(* Logix 5000 project; controller PBS_Perfusion vendor 1 type 14 code 217 rev 32.14; software revision 32.03; part 5 of 27 *)
(* tags used below, declared in another part *)
   ONS : DINT[3];
   P101 : P_VSD;   // Feed Pump
   P103 : P_VSD;   // Conditioned Media Addition Pump
   P104 : P_VSD;   // Recirculation Pump
   P105 : P_VSD;   // Spent Media Pump
   REAL : DINT;

ADD_ON_INSTRUCTION AMP_Update_Jog_Speed   (* revision 1.0 *)
// Applied Motion - Update Jog Speed AOI
// Help:
// The Jog Move AOI is used to start jogging an axis at a specified speed and direction (a negative speed set point implies a CCW direction).
VAR_IN_OUT
   Input : DINT[14]; {required}   // Drive Input Assembly
   Output : DINT[16]; {required}   // Drive Output Assembly
        [0]   // Command Word
        [1]   // Jog Speed (0.25 rev/min)
        [2]   // Jog Acceleration (10 rev/s/s)
        [3]   // Jog Deceleration (10 rev/s/s)
        [4]   // Point-to-Point Velocity (0.25 rev/min)
        [5]   // Point-to-Point Acceleration (10 rev/min/s)
        [6]   // Point-to-Point Deceleration (10 rev/min/s)
        [7]   // Point-to-Point Distance (Motor steps)
        [9]   // (2x ASCII Letters in 16 lower word)
        [10]   // Data/Register 1
        [11]   // Data/Register 2
END_VAR
VAR_INPUT
   RPI : DINT := 100; {visible}   // Drive Connection Request Packet Interval (milliseconds)
   Start : BOOL; {required}   // Start the Relative Move
   Speed : REAL; {required}   // Updated Jog Velocity (rev/min)
END_VAR
VAR_OUTPUT
   Sent : BOOL; {access Read Only, visible}   // Updated Jog Velocity has been sent to drive
   In_Progress : BOOL; {access Read Only, visible}   // Jog Velocity Update in progress
   Done : BOOL; {access Read Only, visible}   // Jog Velocity Update completed without errors
   Error : BOOL; {access Read Only, visible}   // Jog Velocity Update failed to complete - drive not ready or faulted
   State : DINT := 10; {access Read Only}   // Internal state of progress
END_VAR
VAR
   Loc_StatusCode : AMP_Status_Word;
   Loc_CommandOff_Timer : TIMER;   // Timer to make sure command value was 0 before sending a new command
   Loc_CommandOn_Timer : TIMER;   // Timer to make sure command value is set long enough to be sent to drive
   Loc_Input_Assembly : AMP_Input_Assembly_v2; {access None}
   Loc_Start_ONS : BOOL; {access None}
   Loc_AlarmCode : AMP_Alarm_Word; {access None}
END_VAR

ROUTINE Logic   (* ladder *)
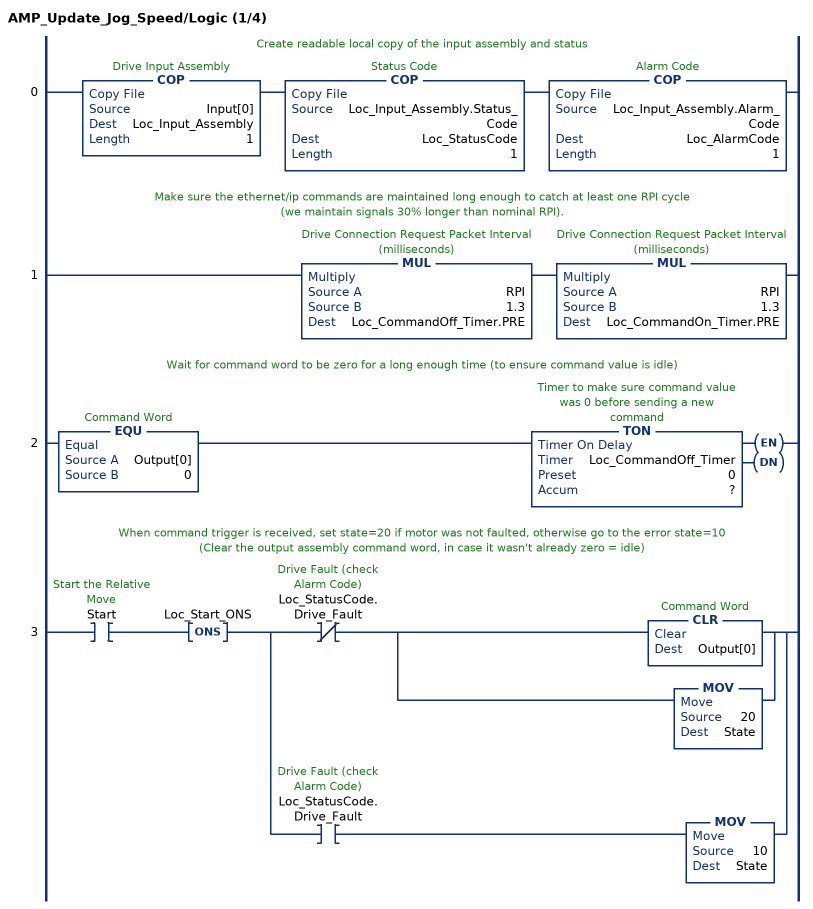
   // Create readable local copy of the input assembly and status
   0: COP(Input[0],Loc_Input_Assembly,1)COP(Loc_Input_Assembly.Status_Code,Loc_StatusCode,1)COP(Loc_Input_Assembly.Alarm_Code,Loc_AlarmCode,1);
   // Make sure the ethernet/ip commands are maintained long enough to catch at least one RPI cycle
   // (we maintain signals 30% longer than nominal RPI).
   1: MUL(RPI,1.3,Loc_CommandOff_Timer.PRE)MUL(RPI,1.3,Loc_CommandOn_Timer.PRE);
   // Wait for command word to be zero for a long enough time (to ensure command value is idle)
   2: EQU(Output[0],0)TON(Loc_CommandOff_Timer,?,?);
   // When command trigger is received, set state=20 if motor was not faulted, otherwise go to the error state=10
   // (Clear the output assembly command word, in case it wasn't already zero = idle)
   3: XIC(Start)ONS(Loc_Start_ONS)[XIO(Loc_StatusCode.Drive_Fault) [CLR(Output[0]) ,MOV(20,State) ] ,XIC(Loc_StatusCode.Drive_Fault) MOV(10,State) ];
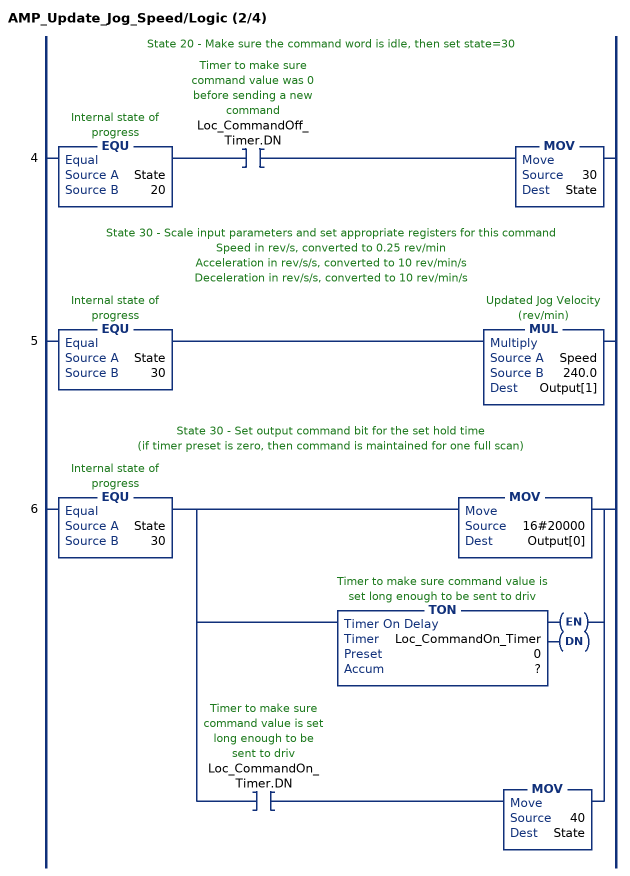
   // State 20 - Make sure the command word is idle, then set state=30
   4: EQU(State,20)XIC(Loc_CommandOff_Timer.DN)MOV(30,State);
   // State 30 - Scale input parameters and set appropriate registers for this command
   // Speed in rev/s, converted to 0.25 rev/min
   // Acceleration in rev/s/s, converted to 10 rev/min/s
   // Deceleration in rev/s/s, converted to 10 rev/min/s
   5: EQU(State,30)MUL(Speed,240.0,Output[1]);
   // State 30 - Set output command bit for the set hold time
   // (if timer preset is zero, then command is maintained for one full scan)
   6: EQU(State,30)[MOV(16#20000,Output[0]) ,TON(Loc_CommandOn_Timer,?,?) ,XIC(Loc_CommandOn_Timer.DN) MOV(40,State) ];
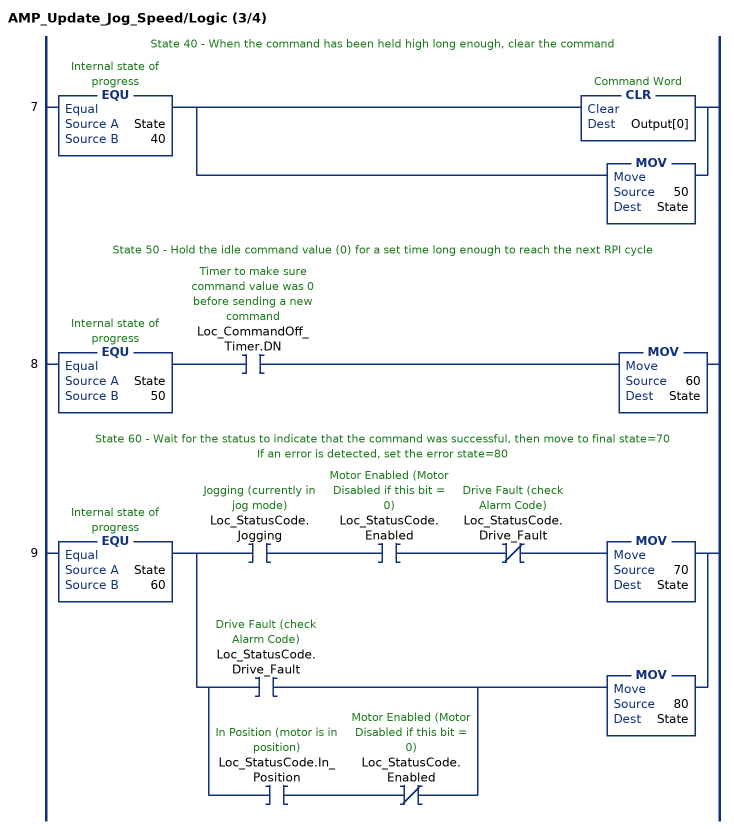
   // State 40 - When the command has been held high long enough, clear the command
   7: EQU(State,40)[CLR(Output[0]) ,MOV(50,State) ];
   // State 50 - Hold the idle command value (0) for a set time long enough to reach the next RPI cycle
   8: EQU(State,50)XIC(Loc_CommandOff_Timer.DN)MOV(60,State);
   // State 60 - Wait for the status to indicate that the command was successful, then move to final state=70
   // If an error is detected, set the error state=80
   9: EQU(State,60)[XIC(Loc_StatusCode.Jogging) XIC(Loc_StatusCode.Enabled) XIO(Loc_StatusCode.Drive_Fault) MOV(70,State) ,[XIC(Loc_StatusCode.Drive_Fault) ,XIC(Loc_StatusCode.In_Position) XIO(Loc_StatusCode.Enabled) ] MOV(80,State) ];
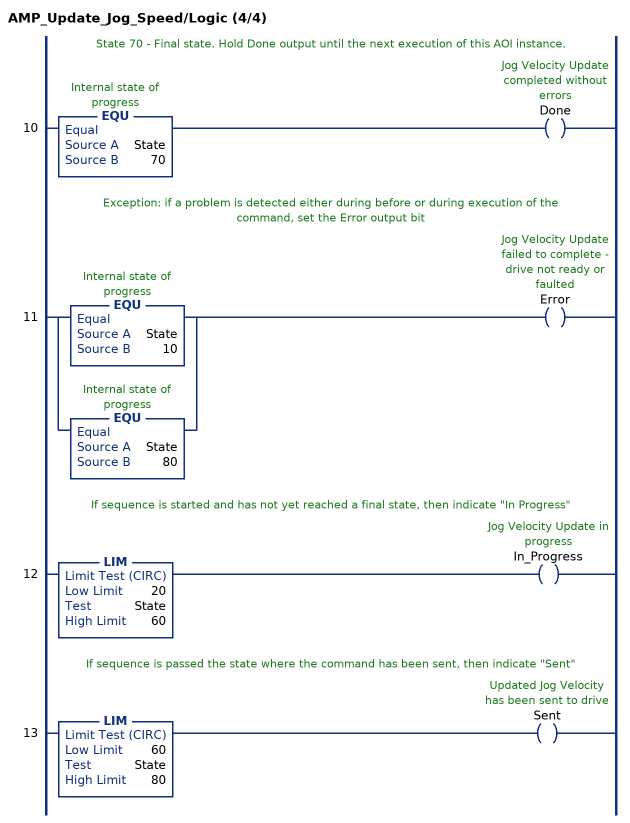
   // State 70 - Final state. Hold Done output until the next execution of this AOI instance.
   10: EQU(State,70)OTE(Done);
   // Exception: if a problem is detected either during before or during execution of the command, set the Error output bit
   11: [EQU(State,10) ,EQU(State,80) ]OTE(Error);
   // If sequence is started and has not yet reached a final state, then indicate "In Progress"
   12: LIM(20,State,60)OTE(In_Progress);
   // If sequence is passed the state where the command has been sent, then indicate "Sent"
   13: LIM(60,State,80)OTE(Sent);
END_ROUTINE
END_ADD_ON_INSTRUCTION

ADD_ON_INSTRUCTION P_AInAdv   (* revision 4.10 .00 Release, vendor Rockwell Automation, ExecutePrescan, ExecuteEnableInFalse *)
// Advanced Analog Input
// Revision note:
// See Instruction Help for a summary of changes, and see 4.10 Release Notes for details.
// Help:
// Copyright © Rockwell Automation, Inc.  All Rights Reserved.
// This Instruction monitors an Analog Input from a flow, level, pressure,
// temperature, or any other analog sensor, and provides:
// *  Scaling, from Input (Raw) to PV (Engineering) Units
// *  High-High, High, Low and Low-Low Status and Alarms, with Gate
//     inputs and configurable on-delay, off-delay and gate delay times
// *  Monitoring of bad/uncertain PV status, floating point exceptions
//     and out-of-range conditions, with PV Fail alarm
// *  Setting of a simulated input signal for process simulation
// *  Capturing of the lowest and highest PV excursion values
// *  Configuration for status thresholds, deadbands and range limits
// *  Maintenance Commands to allow manual override of the input signal (Substitute PV)
// **  Calculation of (filtered) signal rate of change with High Rate of Change alarm
// **  Square Root characterization for flow scaling based on differential-pressure input
// **  Reference (setpoint) value entry and alarms for deviation from reference (high, low)
// ** = advanced capabilities in this instruction
// *  = basic capabilities included in P_AIn (analog input basic) instruction
// Alarms are provided by P_Alarm AOI instances.
// Gating of status provided by P_Gate AOI instances.
// SUMMARY OF CHANGES FROM PREVIOUS VERSION (4.00.01)
// See 4.10 Release Notes for details.
// * Added Control Limits.
// * Added Cfg_HasMoreObj.
// SUMMARY OF CHANGES FROM PREVIOUS VERSION (4.00.00)
// See 4.00 Release Notes for details.
// * Modified handling of SrcQ_IO and SrcQ.
// SUMMARY OF CHANGES FROM PREVIOUS VERSION (3.5-03)
// See 4.00 Release Notes for details.
// * Removed P_Mode, PSet/Val_Owner and related OSets,
//    PSets and Vals.  Thresholds are now Cfgs.
// * Changed Inf_ items to HMI_, and added Cfg_Area for security.
// * Added notify and unack count rollup for Channel object.
// * Added Err_Rate.
// * Changed Out-of-Range limit checks to use raw Input (Inp_PV)
//    instead of scaled PV (Val).  Changing EU scaling will not
//    necessitate changing fail thresholds and deadband.
// * Deleted Cfg_PCmdClear.  All Program Commands are now self-clearing.
// * Aligned ready bit naming with command bit names.
// * All OCmds/MCmds and ORdys/MRdys are now Local Tags.
// * Added Sts_RdyAck and Sts_RdyReset for use by external objects.
// * Removed Err_DB, code ensures Status Deadband configs are always valid.
// * Added configurable decimal places for display on HMI.
VAR_INPUT
   Inp_PV : REAL; {visible}   // Input Signal (process variable) from Sensor
   Inp_PVSrcQ : DINT;   // Input Source and Quality (from Channel object, if available) (enum)
   Inp_PVNotify : DINT;   // Related PV object alarm prio and ack status (enum)
   Inp_PVBad : BOOL;   // 1=PV or I/O Comms Status Bad, 0=OK
   Inp_PVUncertain : BOOL;   // 1=PV Value Not Reliable, 0=OK
   Inp_Sim : BOOL;   // 1=Use simulated PV (Set_SimPV); 0=Use Input (Inp_PV)
   Inp_HiHiGate : ALIAS FOR HiHiGate.Inp_Gate;   // High-High Status Gate, 1=enabled
   Inp_HiGate : ALIAS FOR HiGate.Inp_Gate;   // High Status Gate, 1=enabled
   Inp_LoGate : ALIAS FOR LoGate.Inp_Gate;   // Low Status Gate, 1=enabled
   Inp_LoLoGate : ALIAS FOR LoLoGate.Inp_Gate;   // Low-Low Status Gate, 1=enabled
   Inp_HiRoCGate : ALIAS FOR HiRoCGate.Inp_Gate;   // High Rate of Change Status Gate, 1=enabled
   Inp_HiDevGate : ALIAS FOR HiDevGate.Inp_Gate;   // High Deviation Status Gate, 1=enabled
   Inp_LoDevGate : ALIAS FOR LoDevGate.Inp_Gate;   // Low Deviation Status Gate, 1=enabled
   Inp_FailGate : ALIAS FOR FailGate.Inp_Gate;   // Fail Status Gate, 1=enabled
   Inp_Reset : BOOL;   // 1=Reset all Alarms requiring reset
   Cfg_UseSqRt : BOOL;   // 1=Use Square Root characterization for DP to flow; 0=Linear
   Cfg_HasRoC : BOOL;   // 1=Enables the Rate of Change calc and HiRoC alarm
   Cfg_HasDev : BOOL;   // 1=Enables Reference entry and Deviation calc and alarms
   Cfg_NoSubstPV : BOOL;   // 1=Disallow selection of Substitute PV
   Cfg_HasChanObj : BOOL;   // 1=Tells HMI a Channel object (AIChan, etc.) is used for Inp_PV
   Cfg_HasMoreObj : BOOL;   // 1=Tells HMI an object with more info is available
   Cfg_UseChanSrcQ : BOOL;   // 1=Pass thru connected Channel's SrcQ value, 0=generate SrcQ
   Cfg_PVDecPlcs : DINT := 2;   // Number of decimal places for PV display (0..6)
   Cfg_HasHiHiAlm : ALIAS FOR HiHi.Cfg_Exists;   // 1=High-High Alarm exists and will be checked
   Cfg_HasHiAlm : ALIAS FOR Hi.Cfg_Exists;   // 1=High Alarm exists and will be checked
   Cfg_HasLoAlm : ALIAS FOR Lo.Cfg_Exists;   // 1=Low Alarm exists and will be checked
   Cfg_HasLoLoAlm : ALIAS FOR LoLo.Cfg_Exists;   // 1=Low-Low Alarm exists and will be checked
   Cfg_HasHiRoCAlm : ALIAS FOR HiRoC.Cfg_Exists;   // 1=High Rate of Change Alarm exists and will be checked
   Cfg_HasHiDevAlm : ALIAS FOR HiDev.Cfg_Exists;   // 1=High Deviation Alarm exists and will be checked
   Cfg_HasLoDevAlm : ALIAS FOR LoDev.Cfg_Exists;   // 1=Low Deviation Alarm exists and will be checked
   Cfg_HasFailAlm : ALIAS FOR Fail.Cfg_Exists;   // 1=Analog Input Failure Alarm exists and should be scanned
   Cfg_HiHiResetReqd : ALIAS FOR HiHi.Cfg_ResetReqd;   // 1=Reset required to clear High-High Alarm
   Cfg_HiResetReqd : ALIAS FOR Hi.Cfg_ResetReqd;   // 1=Reset required to clear High Alarm
   Cfg_LoResetReqd : ALIAS FOR Lo.Cfg_ResetReqd;   // 1=Reset required to clear Low Alarm
   Cfg_LoLoResetReqd : ALIAS FOR LoLo.Cfg_ResetReqd;   // 1=Reset required to clear Low-Low Alarm
   Cfg_HiRoCResetReqd : ALIAS FOR HiRoC.Cfg_ResetReqd;   // 1=Reset required to clear High Rate of Change Alarm
   Cfg_HiDevResetReqd : ALIAS FOR HiDev.Cfg_ResetReqd;   // 1=Reset required to clear High Deviation Alarm
   Cfg_LoDevResetReqd : ALIAS FOR LoDev.Cfg_ResetReqd;   // 1=Reset required to clear Low Deviation Alarm
   Cfg_FailResetReqd : ALIAS FOR Fail.Cfg_ResetReqd;   // 1=Reset required to clear Analog InputFailure Alarm
   Cfg_HiHiAckReqd : ALIAS FOR HiHi.Cfg_AckReqd;   // 1=Acknowledge required for High-High Alarm
   Cfg_HiAckReqd : ALIAS FOR Hi.Cfg_AckReqd;   // 1=Acknowledge required for High Alarm
   Cfg_LoAckReqd : ALIAS FOR Lo.Cfg_AckReqd;   // 1=Acknlowledge required for Low Alarm
   Cfg_LoLoAckReqd : ALIAS FOR LoLo.Cfg_AckReqd;   // 1=Acknowledge required for Low-Low Alarm
   Cfg_HiRoCAckReqd : ALIAS FOR HiRoC.Cfg_AckReqd;   // 1=Acknowledge required for High Rate of Change Alarm
   Cfg_HiDevAckReqd : ALIAS FOR HiDev.Cfg_AckReqd;   // 1=Acknowledge required for High Deviation Alarm
   Cfg_LoDevAckReqd : ALIAS FOR LoDev.Cfg_AckReqd;   // 1=Acknowledge required for Low Deviation Alarm
   Cfg_FailAckReqd : ALIAS FOR Fail.Cfg_AckReqd;   // 1=Acknowledge required for Analog Input Failure Alarm
   Cfg_HiHiSeverity : ALIAS FOR HiHi.Cfg_Severity;   // High-High Alarm Severity: 1..250=Low, 251..500=Medium, 501..750=High, 751..1000=Urgent
   Cfg_HiSeverity : ALIAS FOR Hi.Cfg_Severity;   // High Alarm Severity: 1..250=Low, 251..500=Medium, 501..750=High, 751..1000=Urgent
   Cfg_LoSeverity : ALIAS FOR Lo.Cfg_Severity;   // Low Alarm Severity: 1..250=Low, 251..500=Medium, 501..750=High, 751..1000=Urgent
   Cfg_LoLoSeverity : ALIAS FOR LoLo.Cfg_Severity;   // Low-Low Alarm Severity: 1..250=Low, 251..500=Medium, 501..750=High, 751..1000=Urgent
   Cfg_HiRoCSeverity : ALIAS FOR HiRoC.Cfg_Severity;   // High Rate of Change Severity: 1..250=Low, 251..500=Medium, 501..750=High, 751..1000=Urgent
   Cfg_HiDevSeverity : ALIAS FOR HiDev.Cfg_Severity;   // High Deviation Severity: 1..250=Low, 251..500=Medium, 501..750=High, 751..1000=Urgent
   Cfg_LoDevSeverity : ALIAS FOR LoDev.Cfg_Severity;   // Low Deviation Severity: 1..250=Low, 251..500=Medium, 501..750=High, 751..1000=Urgent
   Cfg_FailSeverity : ALIAS FOR Fail.Cfg_Severity;   // Failure Alarm Severity: 1..250=Low, 251..500=Medium, 501..750=High, 751..1000=Urgent
   Cfg_InpRawMin : REAL;   // Input (unscaled) Minimum for Scaling
   Cfg_InpRawMax : REAL := 100.0;   // Input (unscaled) Maximum for Scaling
   Cfg_PVEUMin : REAL;   // PV (Output) Minimum for Scaling to EU
   Cfg_PVEUMax : REAL := 100.0;   // PV (Output) Maximum for Scaling to EU
   Cfg_FiltTC : REAL;   // PV Filter Time Constant (sec), 0.0 = unfiltered
   Cfg_RateTime : REAL := 1.0;   // PV Rate of Change time base (sec) 60=/min, 3600=/hr
   Cfg_Ref : REAL; {visible}   // Analog Reference for Deviation Alarms (EU)
   Cfg_CtrlHiHiLim : REAL := 1.5e+38;   // Current High-High Control Threshold
   Cfg_CtrlHiHiDB : REAL := 1.0;   // High-High Control Deadband (EU)
   Cfg_CtrlHiLim : REAL := 1.5e+38;   // Current High Control Threshold
   Cfg_CtrlHiDB : REAL := 1.0;   // High Control Deadband (EU)
   Cfg_CtrlLoLim : REAL := -1.5e+38;   // Current Low Control Threshold
   Cfg_CtrlLoDB : REAL := 1.0;   // Low Control Deadband (EU)
   Cfg_CtrlLoLoLim : REAL := -1.5e+38;   // Current Low-Low Control Threshold
   Cfg_CtrlLoLoDB : REAL := 1.0;   // Low-Low Control Deadband (EU)
   Cfg_HiHiLim : REAL := 1.5e+38; {visible}   // Current High-High Status Threshold
   Cfg_HiHiDB : REAL := 1.0;   // High-High Status Deadband (EU)
   Cfg_HiHiOnDly : ALIAS FOR HiHiGate.Cfg_OnDly;   // Minimum time above High-High Limit to raise Status (sec)
   Cfg_HiHiOffDly : ALIAS FOR HiHiGate.Cfg_OffDly;   // Minimum time below High-High Limit (minus deadband) to clear Status (sec)
   Cfg_HiHiGateDly : ALIAS FOR HiHiGate.Cfg_GateDly;   // High-High Status Gate Delay (s)
   Cfg_HiLim : REAL := 1.5e+38; {visible}   // Current High Status Threshold
   Cfg_HiDB : REAL := 1.0;   // High Status Deadband (EU)
   Cfg_HiOnDly : ALIAS FOR HiGate.Cfg_OnDly;   // Minimum time above High Limit to raise Status (sec)
   Cfg_HiOffDly : ALIAS FOR HiGate.Cfg_OffDly;   // Minimum time below High Limit (minus deadband) to clear Status (sec)
   Cfg_HiGateDly : ALIAS FOR HiGate.Cfg_GateDly;   // High Status Gate Delay (s)
   Cfg_LoLim : REAL := -1.5e+38; {visible}   // Current Low Status Threshold
   Cfg_LoDB : REAL := 1.0;   // Low Status Deadband (EU)
   Cfg_LoOnDly : ALIAS FOR LoGate.Cfg_OnDly;   // Minimum time below Low Limit to raise Status (sec)
   Cfg_LoOffDly : ALIAS FOR LoGate.Cfg_OffDly;   // Minimum time above Low Limit (plus deadband) to clear Status (sec)
   Cfg_LoGateDly : ALIAS FOR LoGate.Cfg_GateDly;   // Low Status Gate Delay (s)
   Cfg_LoLoLim : REAL := -1.5e+38; {visible}   // Current Low-Low Status Threshold
   Cfg_LoLoDB : REAL := 1.0;   // Low-Low Status Deadband (EU)
   Cfg_LoLoOnDly : ALIAS FOR LoLoGate.Cfg_OnDly;   // Minimum time below Low-Low Limit to raise Status (sec)
   Cfg_LoLoOffDly : ALIAS FOR LoLoGate.Cfg_OffDly;   // Minimum time above Low-Low Limit (plus deadband) to clear Status (sec)
   Cfg_LoLoGateDly : ALIAS FOR LoLoGate.Cfg_GateDly;   // Low-Low Status Gate Delay (s)
   Cfg_HiRoCLim : REAL := 1.5e+38; {visible}   // Current High Rate of Change Status Threshold
   Cfg_HiRoCDB : REAL := 1.0;   // High Rate of Change Status Deadband (EU/rate time)
   Cfg_HiRoCOnDly : ALIAS FOR HiRoCGate.Cfg_OnDly;   // Minimum time above High Rate of Change Limit to raise Status (sec)
   Cfg_HiRoCOffDly : ALIAS FOR HiRoCGate.Cfg_OffDly;   // Minimum time below High Rate of Change Limit (minus deadband) to clear Status (sec)
   Cfg_HiRoCGateDly : ALIAS FOR HiRoCGate.Cfg_GateDly;   // High Rate of Change Status Gate Delay (s)
   Cfg_HiDevLim : REAL := 1.5e+38; {visible}   // Current High Deviation Status Threshold
   Cfg_HiDevDB : REAL := 1.0;   // High Deviation Status Deadband (EU)
   Cfg_HiDevOnDly : ALIAS FOR HiDevGate.Cfg_OnDly;   // Minimum time above High Deviation Limit to raise Status (sec)
   Cfg_HiDevOffDly : ALIAS FOR HiDevGate.Cfg_OffDly;   // Minimum time below High Deviation Limit (minus deadband) to clear Status (sec)
   Cfg_HiDevGateDly : ALIAS FOR HiDevGate.Cfg_GateDly;   // High Deviation Status Gate Delay (s)
   Cfg_LoDevLim : REAL := -1.5e+38; {visible}   // Current Low Deviation Status Threshold
   Cfg_LoDevDB : REAL := 1.0;   // Low Deviation Status Deadband (EU)
   Cfg_LoDevOnDly : ALIAS FOR LoDevGate.Cfg_OnDly;   // Minimum time below Low Deviation Limit to raise Status (sec)
   Cfg_LoDevOffDly : ALIAS FOR LoDevGate.Cfg_OffDly;   // Minimum time above Low Deviation Limit (plus deadband) to clear Status (sec)
   Cfg_LoDevGateDly : ALIAS FOR LoDevGate.Cfg_GateDly;   // Low Deviation Status Gate Delay (s)
   Cfg_FailHiLim : REAL := 103.958336;   // Out-of-Range (fail) High Limit (EU)
   Cfg_FailLoLim : REAL := -2.0833333;   // Out-of-Range (fail) Low Limit (EU)
   Cfg_FailDB : REAL := 0.41666666;   // Out-of-Range (fail) High/Low Deadband (EU)
   Cfg_FailOnDly : ALIAS FOR FailGate.Cfg_OnDly;   // Minimum time Bad or Out of Range to raise Fail Status (sec)
   Cfg_FailOffDly : ALIAS FOR FailGate.Cfg_OffDly;   // Minimum time OK or In Range to clear Fail Status (sec)
   Cfg_FailGateDly : ALIAS FOR FailGate.Cfg_GateDly;   // Fail Status Gate Delay (s)
   MSet_SubstPV : REAL;   // Maintenance-Entered Substitute PV (EU)
   Set_SimPV : REAL;   // PV used in Simulation (Inp_Sim=1) (EU)
   PCmd_ClearCapt : BOOL;   // Program Command to Clear the captured min / max PV excursion values
   PCmd_Reset : BOOL;   // Program Command to Reset all Alarms requiring Reset
   PCmd_HiHiAck : ALIAS FOR HiHi.PCmd_Ack;   // Program Command to Acknowledge High-High Alarm
   PCmd_HiHiSuppress : ALIAS FOR HiHi.PCmd_Suppress;   // Program Command to Suppress High-High Alarm
   PCmd_HiHiUnsuppress : ALIAS FOR HiHi.PCmd_Unsuppress;   // Program Command to Unsuppress High-High Alarm
   PCmd_HiHiUnshelve : ALIAS FOR HiHi.PCmd_Unshelve;   // Program Command to Unshelve High-High Alarm
   PCmd_HiAck : ALIAS FOR Hi.PCmd_Ack;   // Program Command to Acknowledge High Alarm
   PCmd_HiSuppress : ALIAS FOR Hi.PCmd_Suppress;   // Program Command to Suppress High Alarm
   PCmd_HiUnsuppress : ALIAS FOR Hi.PCmd_Unsuppress;   // Program Command to Unsuppress High Alarm
   PCmd_HiUnshelve : ALIAS FOR Hi.PCmd_Unshelve;   // Program Command to Unshelve High Alarm
   PCmd_LoAck : ALIAS FOR Lo.PCmd_Ack;   // Program Command to Acknowledge Low Alarm
   PCmd_LoSuppress : ALIAS FOR Lo.PCmd_Suppress;   // Program Command to Suppress Low Alarm
   PCmd_LoUnsuppress : ALIAS FOR Lo.PCmd_Unsuppress;   // Program Command to Unsuppress Low Alarm
   PCmd_LoUnshelve : ALIAS FOR Lo.PCmd_Unshelve;   // Program Command to Unshelve Low Alarm
   PCmd_LoLoAck : ALIAS FOR LoLo.PCmd_Ack;   // Program Command to Acknowledge Low-Low Alarm
   PCmd_LoLoSuppress : ALIAS FOR LoLo.PCmd_Suppress;   // Program Command to Suppress Low-Low Alarm
   PCmd_LoLoUnsuppress : ALIAS FOR LoLo.PCmd_Unsuppress;   // Program Command to Unsuppress Low-Low Alarm
   PCmd_LoLoUnshelve : ALIAS FOR LoLo.PCmd_Unshelve;   // Program Command to Unshelve Low-Low Alarm
   PCmd_HiRoCAck : ALIAS FOR HiRoC.PCmd_Ack;   // Program Command to Acknowledge High Rate of Change Alarm
   PCmd_HiRoCSuppress : ALIAS FOR HiRoC.PCmd_Suppress;   // Program Command to Suppress High Rate of Change Alarm
   PCmd_HiRoCUnsuppress : ALIAS FOR HiRoC.PCmd_Unsuppress;   // Program Command to Unsuppress High Rate of Change Alarm
   PCmd_HiRoCUnshelve : ALIAS FOR HiRoC.PCmd_Unshelve;   // Program Command to Unshelve High Rate of Change Alarm
   PCmd_HiDevAck : ALIAS FOR HiDev.PCmd_Ack;   // Program Command to Acknowledge High Deviation Alarm
   PCmd_HiDevSuppress : ALIAS FOR HiDev.PCmd_Suppress;   // Program Command to Suppress High Deviation Alarm
   PCmd_HiDevUnsuppress : ALIAS FOR HiDev.PCmd_Unsuppress;   // Program Command to Unsuppress High Deviation Alarm
   PCmd_HiDevUnshelve : ALIAS FOR HiDev.PCmd_Unshelve;   // Program Command to Unshelve High Deviation Alarm
   PCmd_LoDevAck : ALIAS FOR LoDev.PCmd_Ack;   // Program Command to Acknowledge Low Deviation Alarm
   PCmd_LoDevSuppress : ALIAS FOR LoDev.PCmd_Suppress;   // Program Command to Suppress Low Deviation Alarm
   PCmd_LoDevUnsuppress : ALIAS FOR LoDev.PCmd_Unsuppress;   // Program Command to Unsuppress Low Deviation Alarm
   PCmd_LoDevUnshelve : ALIAS FOR LoDev.PCmd_Unshelve;   // Program Command to Unshelve Low Deviation Alarm
   PCmd_FailAck : ALIAS FOR Fail.PCmd_Ack;   // Program Command to Acknowldege Analog Input Failure Alarm
   PCmd_FailSuppress : ALIAS FOR Fail.PCmd_Suppress;   // Program Command to Suppress Analog Input Failure Alarm
   PCmd_FailUnsuppress : ALIAS FOR Fail.PCmd_Unsuppress;   // Program Command to Unsuppress Analog Input Failure Alarm
   PCmd_FailUnshelve : ALIAS FOR Fail.PCmd_Unshelve;   // Program Command to Unshelve Analog Input Failure Alarm
END_VAR
VAR_OUTPUT
   Val : REAL; {access Read Only, visible}   // Analog Input Value (incl. Manual Override, if used)
   Val_InpPV : REAL; {access Read Only, visible}   // Analog Input Value (actual, before Substitute PV selection)
   Val_RoC : REAL; {access Read Only, visible}   // Analog Value Rate of Change (EU/rate time)
   Val_Dev : REAL; {access Read Only, visible}   // Calculated Deviation from Reference (EU)
   Val_PVMinCapt : REAL := 1.5e+38; {access Read Only}   // Captured PV Minimum (excursion) since last cleared
   Val_PVMaxCapt : REAL := -1.5e+38; {access Read Only}   // Captured PV Maximum (excursion) since last cleared
   Val_PVEUMin : REAL; {access Read Only}   // Minimum of scaled range = MIN (Cfg_PVEUMin, Cfg_PVEUMax)
   Val_PVEUMax : REAL := 100.0; {access Read Only}   // Maximum of scaled range = MAX (Cfg_PVEUMin, Cfg_PVEUMax)
   SrcQ_IO : DINT; {access Read Only}   // Source and Quality of primary I/O (enumeration)
   SrcQ : DINT; {access Read Only}   // Source and Quality of primary Val/Sts (enumeration)
   Val_Fault : DINT; {access Read Only}   // Device Fault Status 0=none, 20=Lo, 21=Hi, 22=LoDev, 23=HiDev, 24=LoLo, 25=HiHi, 26=HiRoC 32=Fail, 34=CfgErr
   Val_NotifyAll : DINT; {access Read Only}   // Highest Alarm prio and ack status this object + channel (enum)
   Val_UnackAlmC : DINT; {access Read Only}   // Count of Unacknowledged Alarms
   Sts_SubstPV : BOOL; {access Read Only}   // 1=Using Substitute PV (Input being overridden)
   Sts_PVBad : BOOL; {access Read Only}   // 1=PV Bad quality or Out of Range
   Sts_PVUncertain : BOOL; {access Read Only}   // 1=PV Value is Uncertain (quality)
   Sts_MaintByp : BOOL; {access Read Only}   // 1=A Maintenance Bypass is Active, display icon
   Sts_AlmInh : BOOL; {access Read Only}   // 1=An Alarm is Shelved, Disabled or Suppressed: display icon
   Sts_Err : BOOL; {access Read Only, visible}   // 1=Error in Config: see detail bits for reason
   Err_Raw : BOOL; {access Read Only}   // 1=Error in Config: Raw Input Scaling Min = Max
   Err_EU : BOOL; {access Read Only}   // 1=Error in Config: Scaled EU Min = Max
   Err_Timer : BOOL; {access Read Only}   // 1=Error in Config: On-Delay, Off-Delay, Gate Delay Time Invalid (use 0 to 2147483 s)
   Err_Rate : BOOL; {access Read Only}   // 1=Error in Config: Invalid Rate Time (use 1.0, 60.0, 3600.0, 86400.0...)
   Err_Filt : BOOL; {access Read Only}   // 1=-Error in Config: PV filter params (RateTime, TC)
   Err_Alarm : BOOL; {access Read Only}   // 1=Error in Config: Alarm Min On Time, Shelf Time, Severity
   Sts_RdyReset : ALIAS FOR ORdy_Reset; {access Read Only}   // 1=A latched alarm or shed condition is ready to be reset
   Sts_RdyAck : BOOL; {access Read Only}   // 1=An alarm is ready to be acknowledged
   Sts_CtrlHiHi : BOOL; {access Read Only}   // 1=Analog Input is above High-High Control limit
   Sts_CtrlHi : BOOL; {access Read Only}   // 1=Analog Input is above High Control limit
   Sts_CtrlLo : BOOL; {access Read Only}   // 1=Analog Input is above Low Control limit
   Sts_CtrlLoLo : BOOL; {access Read Only}   // 1=Analog Input is above Low-Low Control limit
   Sts_HiHiCmp : ALIAS FOR HiHiGate.Inp;   // PV High-High comparison result 1=High-High
   Sts_HiHiGate : ALIAS FOR HiHiGate.Sts_Gate; {access Read Only}   // PV High-High Gate Delay Status, 1=done
   Sts_HiHi : ALIAS FOR HiHi.Inp; {visible}   // 1=Analog Input is above High-High limit
   Alm_HiHi : ALIAS FOR HiHi.Alm;   // 1=Analog Input is in High-High Alarm
   Ack_HiHi : ALIAS FOR HiHi.Ack;   // 1=High-High Alarm has been acknowledged
   Sts_HiHiDisabled : ALIAS FOR HiHi.Disabled;   // 1=High-High Alarm has been Disabled by Maintenance
   Sts_HiHiShelved : ALIAS FOR HiHi.Shelved;   // 1=High-High Alarm has been Shelved by Operator
   Sts_HiHiSuppressed : ALIAS FOR HiHi.Suppressed;   // 1=High-High Alarm has been Suppressed by Program
   Sts_HiCmp : ALIAS FOR HiGate.Inp;   // PV High comparison result 1=High
   Sts_HiGate : ALIAS FOR HiGate.Sts_Gate; {access Read Only}   // PV High Gate Delay Status, 1=done
   Sts_Hi : ALIAS FOR Hi.Inp; {visible}   // 1=Analog Input is above High limit
   Alm_Hi : ALIAS FOR Hi.Alm;   // 1=Analog Input is in High Alarm
   Ack_Hi : ALIAS FOR Hi.Ack;   // 1=High Alarm has been acknowledged
   Sts_HiDisabled : ALIAS FOR Hi.Disabled;   // 1=High Alarm has been Disabled by Maintenance
   Sts_HiShelved : ALIAS FOR Hi.Shelved;   // 1=High Alarm has been Shelved by Operator
   Sts_HiSuppressed : ALIAS FOR Hi.Suppressed;   // 1=High Alarm has been Suppressed by Program
   Sts_LoCmp : ALIAS FOR LoGate.Inp;   // PV Low comparison result 1=Low
   Sts_LoGate : ALIAS FOR LoGate.Sts_Gate; {access Read Only}   // PV Low Gate Delay Status, 1=done
   Sts_Lo : ALIAS FOR Lo.Inp; {visible}   // 1=Analog Input is below Low limit
   Alm_Lo : ALIAS FOR Lo.Alm;   // 1=Analog Input is in Low Alarm
   Ack_Lo : ALIAS FOR Lo.Ack;   // 1=Low Alarm has been acknowledged
   Sts_LoDisabled : ALIAS FOR Lo.Disabled;   // 1=Low Alarm has been Disabled by Maintenance
   Sts_LoShelved : ALIAS FOR Lo.Shelved;   // 1=Low Alarm has been Shelved by Operator
   Sts_LoSuppressed : ALIAS FOR Lo.Suppressed;   // 1=Low Alarm has been Suppressed by Program
   Sts_LoLoCmp : ALIAS FOR LoLoGate.Inp;   // PV Low-Low comparison result 1=Low-Low
   Sts_LoLoGate : ALIAS FOR LoLoGate.Sts_Gate; {access Read Only}   // PV Low-Low Gate Delay Status, 1=done
   Sts_LoLo : ALIAS FOR LoLo.Inp; {visible}   // 1=Analog Input is below Low-Low limit
   Alm_LoLo : ALIAS FOR LoLo.Alm;   // 1=Analog Input is in Low-Low Alarm
   Ack_LoLo : ALIAS FOR LoLo.Ack;   // 1=Low-Low Alarm has been acknowledged
   Sts_LoLoDisabled : ALIAS FOR LoLo.Disabled;   // 1=Low-Low Alarm has been Disabled by Maintenance
   Sts_LoLoShelved : ALIAS FOR LoLo.Shelved;   // 1=Low-Low Alarm has been Shelved by Operator
   Sts_LoLoSuppressed : ALIAS FOR LoLo.Suppressed;   // 1=Low Low Alarm has been Suppressed by Program
   Sts_HiRoCCmp : ALIAS FOR HiRoCGate.Inp;   // PV High Rate of Change comparison result 1=High
   Sts_HiRoCGate : ALIAS FOR HiRoCGate.Sts_Gate; {access Read Only}   // PV High Rate of Change Gate Delay Status, 1=done
   Sts_HiRoC : ALIAS FOR HiRoC.Inp; {visible}   // 1=Analog Input Rate of Change is above High limit
   Alm_HiRoC : ALIAS FOR HiRoC.Alm;   // 1=Analog Input Rate of Change is in High Alarm
   Ack_HiRoC : ALIAS FOR HiRoC.Ack;   // 1=High Rate of Change Alarm has been acknowledged
   Sts_HiRoCDisabled : ALIAS FOR HiRoC.Disabled;   // 1=High Rate of Change Alarm has been Disabled by Maintenance
   Sts_HiRoCShelved : ALIAS FOR HiRoC.Shelved;   // 1=High Rate of Change Alarm has been Shelved by Operator
   Sts_HiRoCSuppressed : ALIAS FOR HiRoC.Suppressed;   // 1=High Rate of Change Alarm has been Suppressed by Program
   Sts_HiDevCmp : ALIAS FOR HiDevGate.Inp;   // PV High Deviation comparison result 1=Dev High
   Sts_HiDevGate : ALIAS FOR HiDevGate.Sts_Gate; {access Read Only}   // PV High Deviation Gate Delay Status, 1=done
   Sts_HiDev : ALIAS FOR HiDev.Inp; {visible}   // 1=Analog Input Deviation is above High limit
   Alm_HiDev : ALIAS FOR HiDev.Alm;   // 1=Analog Input Deviation is in High Alarm
   Ack_HiDev : ALIAS FOR HiDev.Ack;   // 1=High Deviation Alarm has been acknowledged
   Sts_HiDevDisabled : ALIAS FOR HiDev.Disabled;   // 1=High Deviation Alarm has been Disabled by Maintenance
   Sts_HiDevShelved : ALIAS FOR HiDev.Shelved;   // 1=High Deviation Alarm has been Shelved by Operator
   Sts_HiDevSuppressed : ALIAS FOR HiDev.Suppressed;   // 1=High Deviation Alarm has been Suppressed by Program
   Sts_LoDevCmp : ALIAS FOR LoDevGate.Inp;   // PV Low Deviation comparison result 1=Dev Low
   Sts_LoDevGate : ALIAS FOR LoDevGate.Sts_Gate; {access Read Only}   // PV Low Deviation Gate Delay Status, 1=done
   Sts_LoDev : ALIAS FOR LoDev.Inp; {visible}   // 1=Analog Input Deviation is below Low limit
   Alm_LoDev : ALIAS FOR LoDev.Alm;   // 1=Analog Input Deviation is in Low Alarm
   Ack_LoDev : ALIAS FOR LoDev.Ack;   // 1=Low Deviation Alarm has been acknowledged
   Sts_LoDevDisabled : ALIAS FOR LoDev.Disabled;   // 1=Low Deviation Alarm has been Disabled by Maintenance
   Sts_LoDevShelved : ALIAS FOR LoDev.Shelved;   // 1=Low Deviation Alarm has been Shelved by Operator
   Sts_LoDevSuppressed : ALIAS FOR LoDev.Suppressed;   // 1=Low Deviation Alarm has been Suppressed by Program
   Sts_FailCmp : ALIAS FOR FailGate.Inp;   // PV Fail comparison result 1=Out of Range
   Sts_FailGate : ALIAS FOR FailGate.Sts_Gate; {access Read Only}   // PV Fail Gate Delay Status, 1=done
   Sts_Fail : ALIAS FOR Fail.Inp; {visible}   // 1=Analog Input is Out of Range or PV Bad
   Alm_Fail : ALIAS FOR Fail.Alm;   // 1=Analog Input Failure Alarm (Bad or Out of Range)
   Ack_Fail : ALIAS FOR Fail.Ack;   // 1=Analog Input Failure Alarm has been acknowledged
   Sts_FailDisabled : ALIAS FOR Fail.Disabled;   // 1=Analog input Failure Alarm has been Disabled by Maintenance
   Sts_FailShelved : ALIAS FOR Fail.Shelved;   // 1=Analog Input Failure Alarm has been Shelved by Operator
   Sts_FailSuppressed : ALIAS FOR Fail.Suppressed;   // 1=Analog Input Failure Alarm has been Suppressed by Program
   P_AInAdv : BOOL;   // Unique Parameter Name for auto - discovery
END_VAR
VAR
   LoLo : P_Alarm := (Cfg_AckReqd := 1, Cfg_AllowShelve := 1, Cfg_AllowDisable := 1, Cfg_Severity := 750, Cfg_AlmMinOnT := 5, PCfg_AllowExist := 1, Ack := 1);   // Low-Low Alarm
   Lo : P_Alarm := (Cfg_AckReqd := 1, Cfg_AllowShelve := 1, Cfg_AllowDisable := 1, Cfg_Severity := 500, Cfg_AlmMinOnT := 5, PCfg_AllowExist := 1, Ack := 1);   // Low Alarm
   Hi : P_Alarm := (Cfg_AckReqd := 1, Cfg_AllowShelve := 1, Cfg_AllowDisable := 1, Cfg_Severity := 500, Cfg_AlmMinOnT := 5, PCfg_AllowExist := 1, Ack := 1);   // High Alarm
   HiHi : P_Alarm := (Cfg_AckReqd := 1, Cfg_AllowShelve := 1, Cfg_AllowDisable := 1, Cfg_Severity := 750, Cfg_AlmMinOnT := 5, PCfg_AllowExist := 1, Ack := 1);   // High-High Alarm
   Cfg_EU : STRING_8 := '%';   // Engineering Units for display on HMI
   Cfg_Tag : STRING_20 := 'P_AinAdv';   // Tagname for display on HMI
   Cfg_Label : STRING_20 := 'Analog Input';   // Label for graphic symbol displayed on HMI
   Cfg_Desc : STRING_40 := 'Advanced Analog Input';   // Description for display on HMI
   Fail : P_Alarm := (Cfg_AckReqd := 1, Cfg_AllowShelve := 1, Cfg_AllowDisable := 1, Cfg_Severity := 1000, Cfg_AlmMinOnT := 5, PCfg_AllowExist := 1, Ack := 1);   // Analog Input Failure Alarm (bad quality or out of range)
   Wrk_Notify : DINT; {access None}   // Buffer for building Val_Notify
   HMI_Tab : SINT;   // Tab to display (FTView ME)
   Wrk_Fault : DINT; {access None}   // Buffer for building Val_Fault
   Wrk_SrcQ : DINT; {access None}   // Register for building Source / Quality enumeration
   Wrk_SubstPV : BOOL; {access None}   // Internal flag: Using Substitute PV
   Wrk_PVSq : REAL; {access None}   // Square of PV, for square root characterization
   Wrk_EUMinSq : REAL; {access None}   // Square of EU Min, for square root characterization
   Wrk_EUMaxSq : REAL; {access None}   // Square of EU Max, for square root characterization
   Wrk_UnfiltPV : REAL; {access None}   // Unfiltered PV, input to 1st order filter
   Wrk_ScanTime : REAL; {access None}   // Time since this instance was last scanned
   Wrk_FiltPV : REAL; {access None}   // Filtered PV
   Wrk_RoC : REAL; {access None}   // Calculated Rate of Change of PV
   Wrk_PrevPV : REAL; {access None}   // Previous scan's value of Filtered PV
   LoDev : P_Alarm := (Cfg_AckReqd := 1, Cfg_AllowShelve := 1, Cfg_AllowDisable := 1, Cfg_Severity := 500, Cfg_AlmMinOnT := 5, PCfg_AllowExist := 1, Ack := 1);   // Low Deviation Alarm
   HiDev : P_Alarm := (Cfg_AckReqd := 1, Cfg_AllowShelve := 1, Cfg_AllowDisable := 1, Cfg_Severity := 500, Cfg_AlmMinOnT := 5, PCfg_AllowExist := 1, Ack := 1);   // High Deviation Alarm
   HiRoC : P_Alarm := (Cfg_AckReqd := 1, Cfg_AllowShelve := 1, Cfg_AllowDisable := 1, Cfg_Severity := 500, Cfg_AlmMinOnT := 5, PCfg_AllowExist := 1, Ack := 1);   // High Rate of Change Alarm
   Wrk_ScanT : TIMER := (PRE := 2147483647); {access None}   // Scan Timer (milliseconds, always runs)
   Wrk_Alpha : REAL; {access None}   // Filter multiplier = (1 / (1+TC/dT) )
   Wrk_ValidONS : BOOL; {access None}   // Selected PV goes from Infinite or Not a Number to VALID
   Wrk_InpInfNaN : BOOL; {access None}   // Input (Inp_PV or Set_SimPV) Infinite or Not a Number
   Wrk_InpDINT : DINT; {access None}   // Input REAL bit pattern as a DINT (check for Inf/NaN)
   Wrk_SelPVDINT : DINT; {access None}   // Selected PV check for Infinite or Non A Number
   Wrk_SelPVInfNaN : BOOL; {access None}   // Selected PV (Input or Substitute) is Infinite or NaN
   HMI_Type : STRING_16 := 'P_AInAdv'; {access Read Only}   // Must contain AOI name, used for HMI and Information S/W
   Wrk_HiRoC : BOOL; {access None}   // Internal flag: High Rate of Change Status
   Wrk_LoDev : BOOL; {access None}   // Internal flag: Low Deviation Status
   Wrk_HiDev : BOOL; {access None}   // Internal flag: High Deviation Status
   Wrk_Fail : BOOL; {access None}   // Internal flag: Fail Status
   Wrk_LoLo : BOOL; {access None}   // Internal flag: Low-Low Status
   Wrk_Lo : BOOL; {access None}   // Internal flag: Low Status
   Wrk_HiHi : BOOL; {access None}   // Internal flag: High-High Status
   Wrk_Hi : BOOL; {access None}   // Internal flag: High Status
   LoDevGate : P_Gate := (Inp_Gate := 1);   // Low Deviation Alarm Gate / Delay Block
   HiRoCGate : P_Gate := (Inp_Gate := 1);   // High Rate of Change Alarm Gate / Delay Block
   HiDevGate : P_Gate := (Inp_Gate := 1);   // High Deviation Alarm Gate / Delay Block
   LoLoGate : P_Gate := (Inp_Gate := 1);   // Low-Low Alarm Gate / Delay Block
   LoGate : P_Gate := (Inp_Gate := 1);   // Low Alarm Gate / Delay Block
   HiHiGate : P_Gate := (Inp_Gate := 1);   // High-High Alarm Gate / Delay Block
   HiGate : P_Gate := (Inp_Gate := 1);   // High Alarm Gate / Delay Block
   FailGate : P_Gate := (Inp_Gate := 1);   // Fail Alarm Gate / Delay Block
   HMI_Lib : STRING_12 := 'RA-BAS'; {access Read Only}   // Display Library for Faceplate call-up
   Cfg_Area : STRING_Area := 'area01';   // Process Area for security
   Wrk_UnackAlmC : DINT; {access None}   // Buffer for building Val_UnackAlmC
   Val_Notify : DINT; {access Read Only}   // Highest Alarm prio and ack status this object only (enum)
   OCmd_ResetAckAll : BOOL;   // Operator Command to Reset and Acknowledge all Alarms
   OCmd_Reset : BOOL;   // Operator Command to Reset all Alarms requiring Reset
   OCmd_ClearCapt : BOOL;   // Operator Command to Clear the captured min / max PV excursion values
   MCmd_InpPV : BOOL;   // Maintenance Command to use Input PV (normal)
   MCmd_SubstPV : BOOL;   // Maintenance Command to use Substitute PV (override input)
   ORdy_ResetAckAll : BOOL; {access Read Only}   // 1=Ready for OCmd_ResetAckAll (enables HMI button)
   ORdy_Reset : BOOL; {access Read Only}   // 1=Ready for OCmd_Reset (enables HMI button)
   MRdy_InpPV : BOOL; {access Read Only}   // 1=Ready for MCmd_InpPV (enables HMI button)
   MRdy_SubstPV : BOOL; {access Read Only}   // 1=Ready for MCmd_SubstPV (enables HMI button)
   Wrk_RawPV : REAL; {access None}   // Value of raw PV to be used for Out of Range checking
END_VAR

ROUTINE EnableInFalse   (* ladder *)
// Off-Scan: no Val update or alarm checking.  PV Bad Quality ("stale") is asserted.
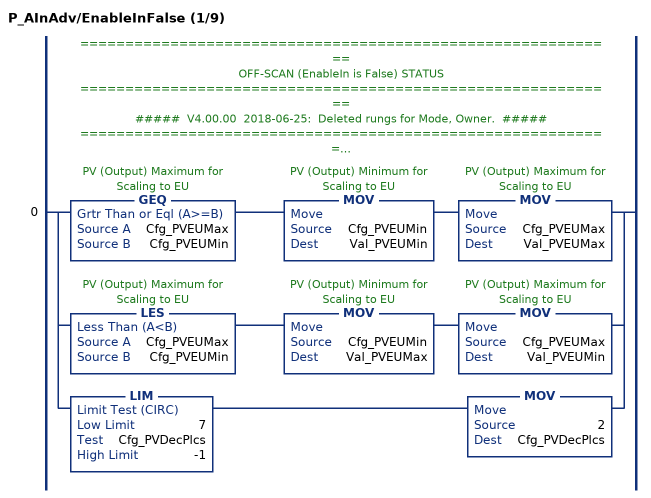
   // ============================================================
   // OFF-SCAN (EnableIn is False) STATUS
   // ============================================================
   // #####  V4.00.00  2018-06-25:  Deleted rungs for Mode, Owner.  #####
   // ============================================================
   // CONFIGURATION
   // ============================================================
   // This rung publishes the Values for the scaled range.
   // If this instruction is reverse scaled by reversing the scaled (EU) min and max configurations,
   // the values are swapped so the the EUMax Value is always greater than the EUMin Value.
   // This makes the HMI bargraph and trend coding easier, and provides values
   // that can be pinned to the configuration of a PID, so the AIn and PID ranges are in lockstep.
   // #####  V4.00.00  2018-06-25:  Added configurable decimal places for display on HMI.  #####
   0: [GEQ(Cfg_PVEUMax,Cfg_PVEUMin) MOV(Cfg_PVEUMin,Val_PVEUMin) MOV(Cfg_PVEUMax,Val_PVEUMax) ,LES(Cfg_PVEUMax,Cfg_PVEUMin) MOV(Cfg_PVEUMin,Val_PVEUMax) MOV(Cfg_PVEUMax,Val_PVEUMin) ,LIM(7,Cfg_PVDecPlcs,-1) MOV(2,Cfg_PVDecPlcs) ];
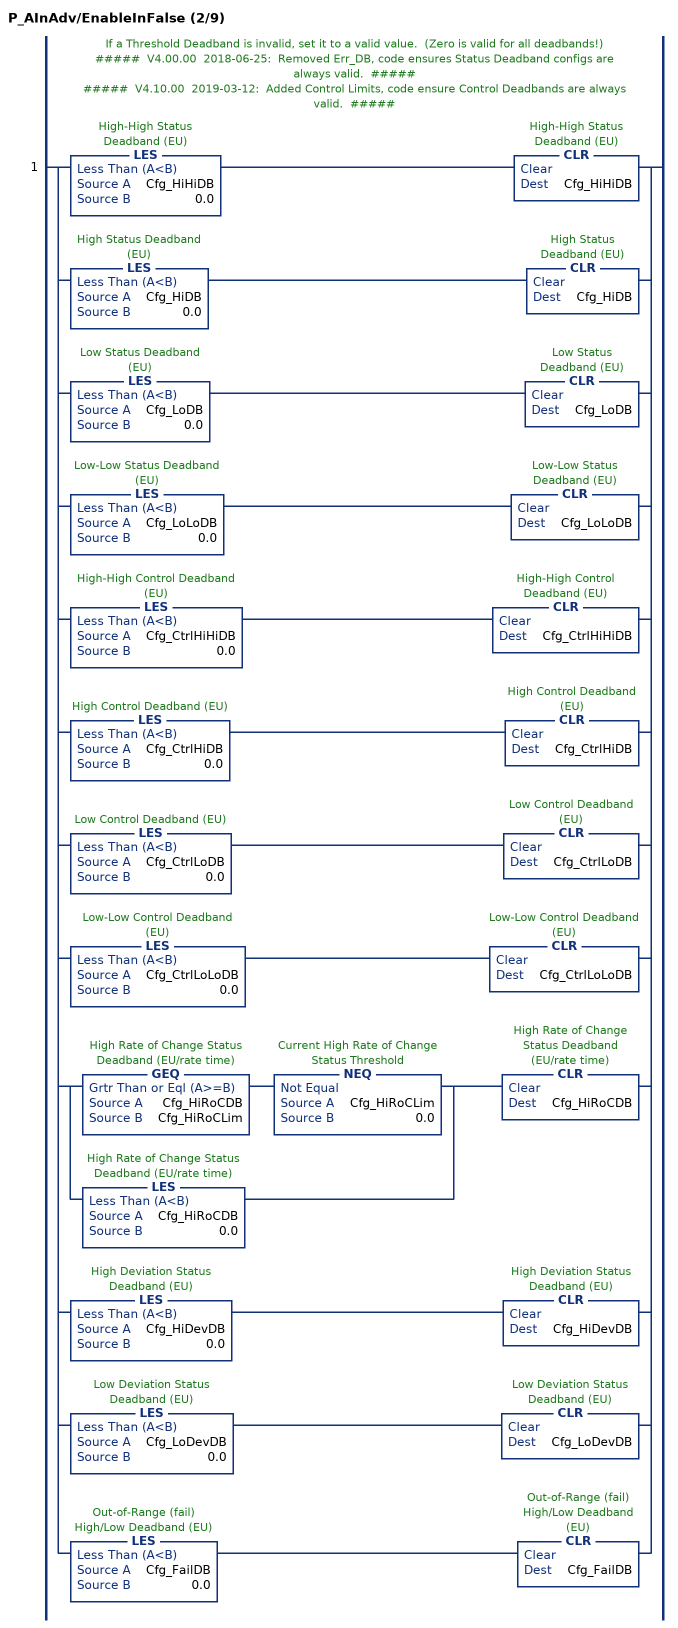
   // If a Threshold Deadband is invalid, set it to a valid value.  (Zero is valid for all deadbands!)
   // #####  V4.00.00  2018-06-25:  Removed Err_DB, code ensures Status Deadband configs are always valid.  #####
   // #####  V4.10.00  2019-03-12:  Added Control Limits, code ensure Control Deadbands are always valid.  #####
   1: [LES(Cfg_HiHiDB,0.0) CLR(Cfg_HiHiDB) ,LES(Cfg_HiDB,0.0) CLR(Cfg_HiDB) ,LES(Cfg_LoDB,0.0) CLR(Cfg_LoDB) ,LES(Cfg_LoLoDB,0.0) CLR(Cfg_LoLoDB) ,LES(Cfg_CtrlHiHiDB,0.0) CLR(Cfg_CtrlHiHiDB) ,LES(Cfg_CtrlHiDB,0.0) CLR(Cfg_CtrlHiDB) ,LES(Cfg_CtrlLoDB,0.0) CLR(Cfg_CtrlLoDB) ,LES(Cfg_CtrlLoLoDB,0.0) CLR(Cfg_CtrlLoLoDB) ,[GEQ(Cfg_HiRoCDB,Cfg_HiRoCLim) NEQ(Cfg_HiRoCLim,0.0) ,LES(Cfg_HiRoCDB,0.0) ] CLR(Cfg_HiRoCDB) ,LES(Cfg_HiDevDB,0.0) CLR(Cfg_HiDevDB) ,LES(Cfg_LoDevDB,0.0) CLR(Cfg_LoDevDB) ,LES(Cfg_FailDB,0.0) CLR(Cfg_FailDB) ];
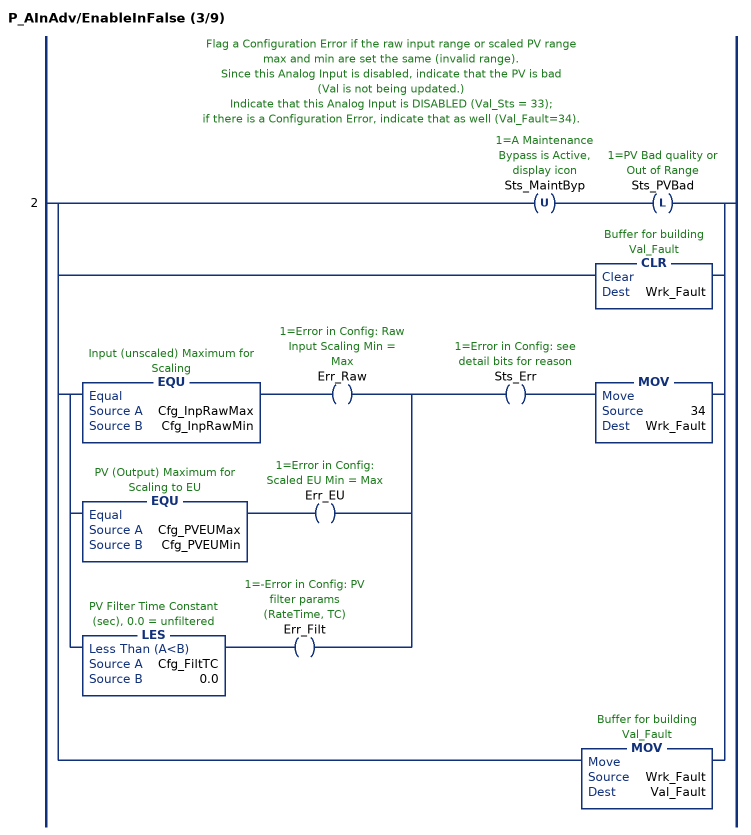
   // Flag a Configuration Error if the raw input range or scaled PV range
   // max and min are set the same (invalid range).
   // Since this Analog Input is disabled, indicate that the PV is bad
   // (Val is not being updated.)
   // Indicate that this Analog Input is DISABLED (Val_Sts = 33);
   // if there is a Configuration Error, indicate that as well (Val_Fault=34).
   2: [OTU(Sts_MaintByp) OTL(Sts_PVBad) ,CLR(Wrk_Fault) ,[EQU(Cfg_InpRawMax,Cfg_InpRawMin) OTE(Err_Raw) ,EQU(Cfg_PVEUMax,Cfg_PVEUMin) OTE(Err_EU) ,LES(Cfg_FiltTC,0.0) OTE(Err_Filt) ] OTE(Sts_Err) MOV(34,Wrk_Fault) ,MOV(Wrk_Fault,Val_Fault) ];
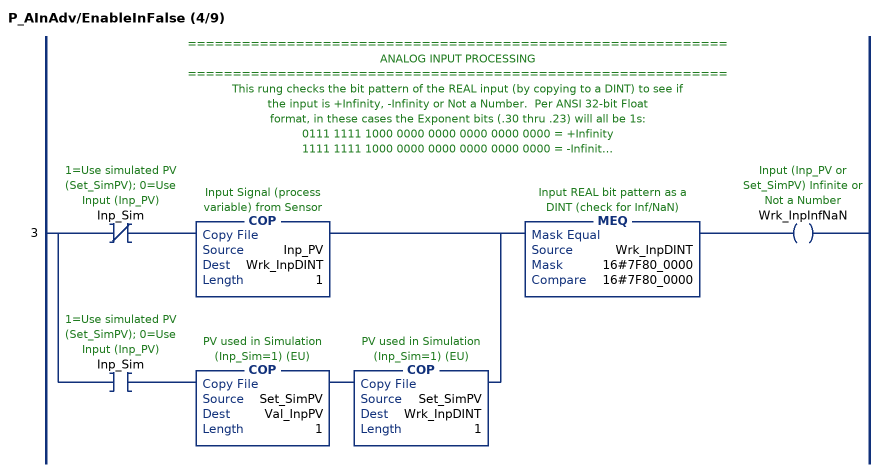
   // ============================================================
   // ANALOG INPUT PROCESSING
   // ============================================================
   // This rung checks the bit pattern of the REAL input (by copying to a DINT) to see if
   // the input is +Infinity, -Infinity or Not a Number.  Per ANSI 32-bit Float
   // format, in these cases the Exponent bits (.30 thru .23) will all be 1s:
   // 0111 1111 1000 0000 0000 0000 0000 0000 = +Infinity
   // 1111 1111 1000 0000 0000 0000 0000 0000 = -Infinity
   // x111 1111 1xxx xxxx xxxx xxxx xxxx xxxx = Not a Number
   3: [XIO(Inp_Sim) COP(Inp_PV,Wrk_InpDINT,1) ,XIC(Inp_Sim) COP(Set_SimPV,Val_InpPV,1) COP(Set_SimPV,Wrk_InpDINT,1) ]MEQ(Wrk_InpDINT,16#7F80_0000,16#7F80_0000)OTE(Wrk_InpInfNaN);
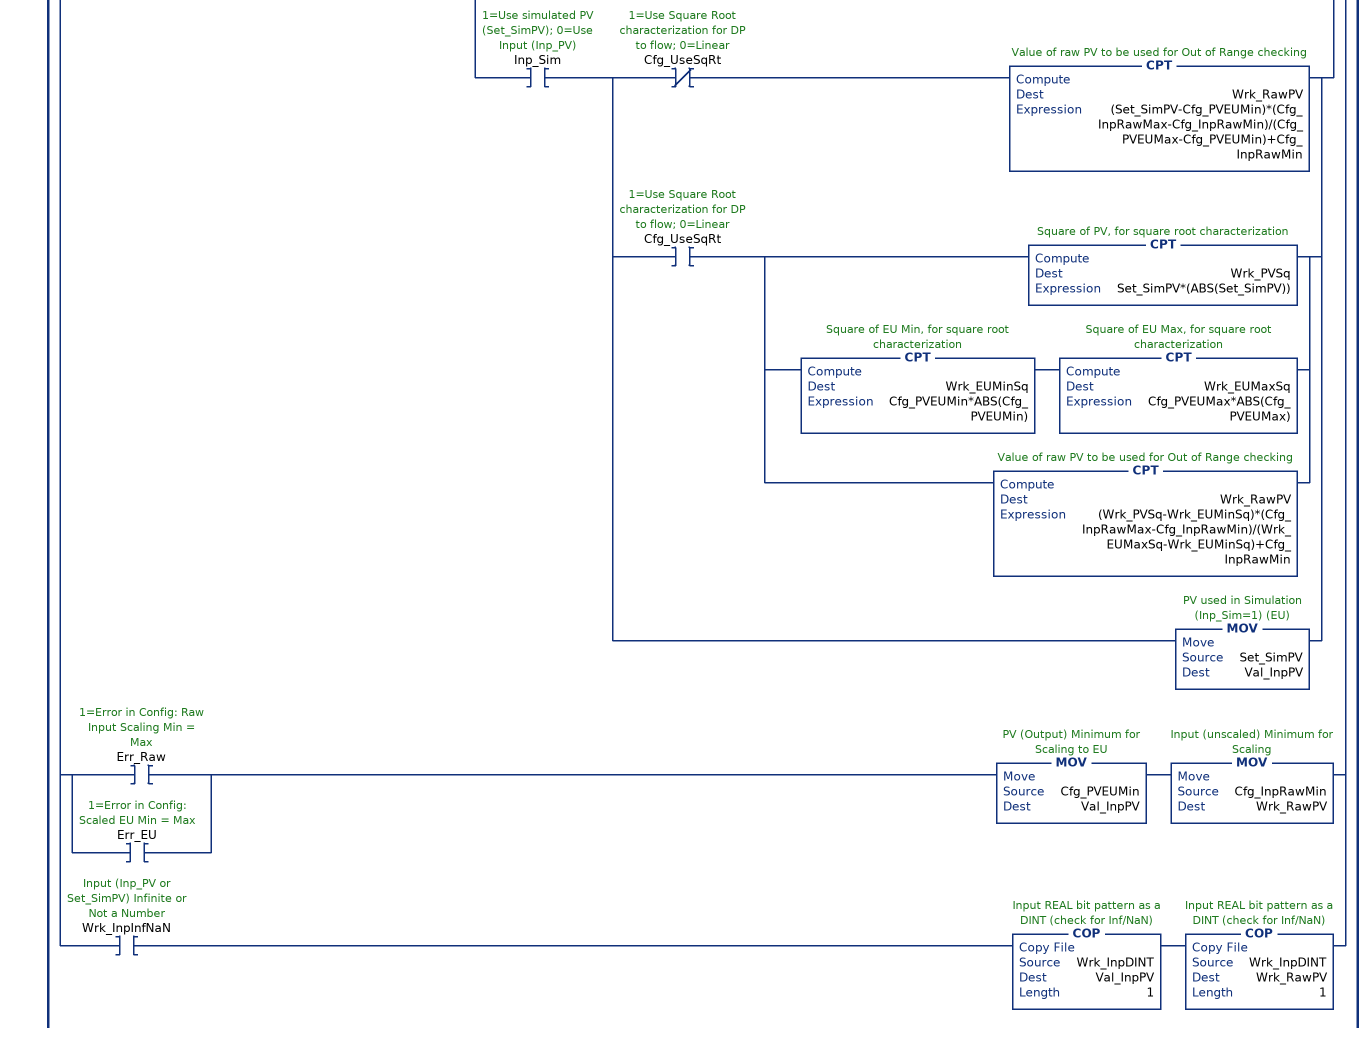
   // The Process Variable Value (Val_PV) shows the selected input,
   // regardless of Mode, EVEN WHEN EnableIn IS FALSE!
   // Here's where we select the input or the substitue PV,
   // and for the input PV, do the scaling to Engineering Units.
   // Scale to the squares of the EUMax and EUMin, then take the Square Root,
   // if the Square Root characterization is selected.  (This must work even for non-zero-based
   // inputs, say, +/- 20" WC, and show +/- flow, scaled on a square root curve each side of zero!)
   // If Square Root characterization is not selected, just do linear scaling.
   4: [XIO(Err_Raw) XIO(Err_EU) XIO(Wrk_InpInfNaN) [XIO(Inp_Sim) [XIO(Cfg_UseSqRt) CPT(Val_InpPV,(Inp_PV-Cfg_InpRawMin)*(Cfg_PVEUMax-Cfg_PVEUMin)/(Cfg_InpRawMax-Cfg_InpRawMin)+Cfg_PVEUMin) ,XIC(Cfg_UseSqRt) [CPT(Wrk_EUMinSq,Cfg_PVEUMin*ABS(Cfg_PVEUMin)) CPT(Wrk_EUMaxSq,Cfg_PVEUMax*ABS(Cfg_PVEUMax)) ,CPT(Wrk_PVSq,(Inp_PV-Cfg_InpRawMin)*(Wrk_EUMaxSq-Wrk_EUMinSq)/(Cfg_InpRawMax-Cfg_InpRawMin)+Wrk_EUMinSq) ,LES(Wrk_PVSq,0.0) CPT(Val_InpPV,-SQR(-Wrk_PVSq)) ,GEQ(Wrk_PVSq,0.0) SQR(Wrk_PVSq,Val_InpPV) ] ,MOV(Inp_PV,Wrk_RawPV) ] ,XIC(Inp_Sim) [XIO(Cfg_UseSqRt) CPT(Wrk_RawPV,(Set_SimPV-Cfg_PVEUMin)*(Cfg_InpRawMax-Cfg_InpRawMin)/(Cfg_PVEUMax-Cfg_PVEUMin)+Cfg_InpRawMin) ,XIC(Cfg_UseSqRt) [CPT(Wrk_PVSq,Set_SimPV*(ABS(Set_SimPV))) ,CPT(Wrk_EUMinSq,Cfg_PVEUMin*ABS(Cfg_PVEUMin)) CPT(Wrk_EUMaxSq,Cfg_PVEUMax*ABS(Cfg_PVEUMax)) ,CPT(Wrk_RawPV,(Wrk_PVSq-Wrk_EUMinSq)*(Cfg_InpRawMax-Cfg_InpRawMin)/(Wrk_EUMaxSq-Wrk_EUMinSq)+Cfg_InpRawMin) ] ,MOV(Set_SimPV,Val_InpPV) ] ] ,[XIC(Err_Raw) ,XIC(Err_EU) ] MOV(Cfg_PVEUMin,Val_InpPV) MOV(Cfg_InpRawMin,Wrk_RawPV) ,XIC(Wrk_InpInfNaN) COP(Wrk_InpDINT,Val_InpPV,1) COP(Wrk_InpDINT,Wrk_RawPV,1) ];
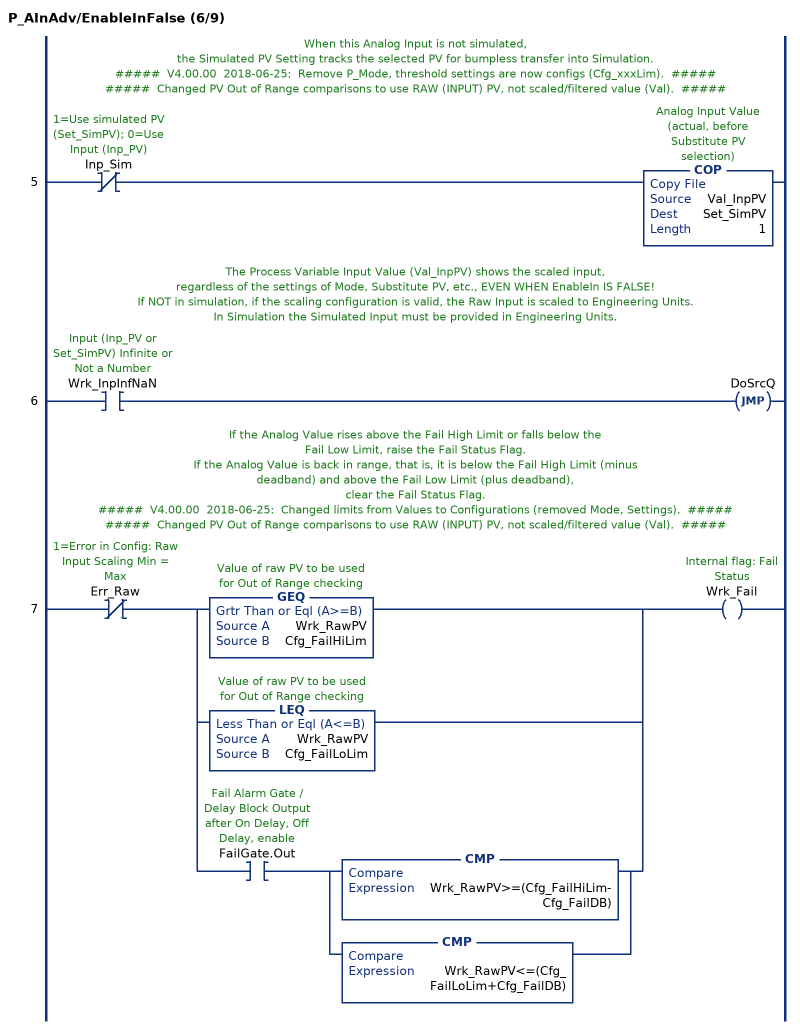
   // When this Analog Input is not simulated,
   // the Simulated PV Setting tracks the selected PV for bumpless transfer into Simulation.
   // #####  V4.00.00  2018-06-25:  Remove P_Mode, threshold settings are now configs (Cfg_xxxLim).  #####
   // #####  Changed PV Out of Range comparisons to use RAW (INPUT) PV, not scaled/filtered value (Val).  #####
   5: XIO(Inp_Sim)COP(Val_InpPV,Set_SimPV,1);
   // The Process Variable Input Value (Val_InpPV) shows the scaled input,
   // regardless of the settings of Mode, Substitute PV, etc., EVEN WHEN EnableIn IS FALSE!
   // If NOT in simulation, if the scaling configuration is valid, the Raw Input is scaled to Engineering Units.
   // In Simulation the Simulated Input must be provided in Engineering Units.
   6: XIC(Wrk_InpInfNaN)JMP(DoSrcQ);
   // If the Analog Value rises above the Fail High Limit or falls below the
   // Fail Low Limit, raise the Fail Status Flag.
   // If the Analog Value is back in range, that is, it is below the Fail High Limit (minus
   // deadband) and above the Fail Low Limit (plus deadband),
   // clear the Fail Status Flag.
   // #####  V4.00.00  2018-06-25:  Changed limits from Values to Configurations (removed Mode, Settings).  #####
   // #####  Changed PV Out of Range comparisons to use RAW (INPUT) PV, not scaled/filtered value (Val).  #####
   7: XIO(Err_Raw)[[GEQ(Wrk_RawPV,Cfg_FailHiLim) ,LEQ(Wrk_RawPV,Cfg_FailLoLim) ] ,XIC(FailGate.Out) [CMP(Wrk_RawPV>=(Cfg_FailHiLim-Cfg_FailDB)) ,CMP(Wrk_RawPV<=(Cfg_FailLoLim+Cfg_FailDB)) ] ]OTE(Wrk_Fail);
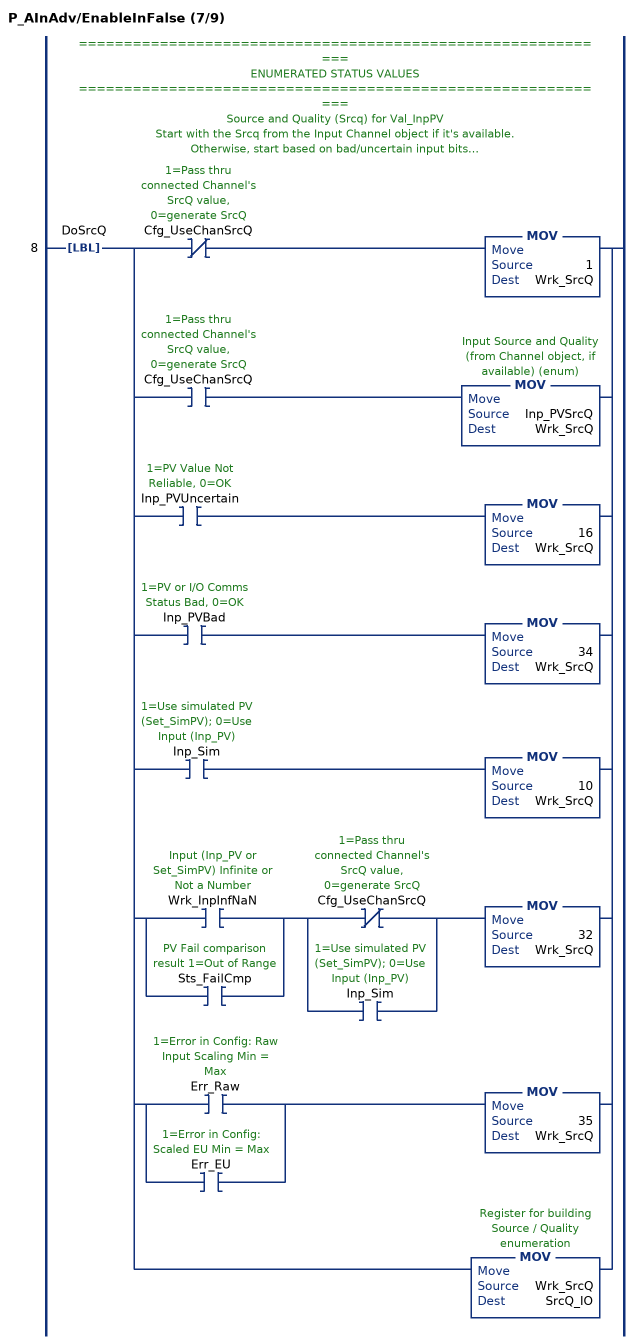
   // ============================================================
   // ENUMERATED STATUS VALUES
   // ============================================================
   // Source and Quality (Srcq) for Val_InpPV
   // Start with the Srcq from the Input Channel object if it's available.
   // Otherwise, start based on bad/uncertain input bits.
   // 0 = Good: live, confirmed good;   1 = Good: live, assumed good;
   // 2 = Good: no feedback, assumed good;   8 = Test: Simulated;   9 = Test: Loopback;
   // 10 = Test: Manually Entered;   16 = Uncertain: Live, off-spec;
   // 17 = Uncertain, Substituted at Device / Bus;   18 = Uncertain, Substituted at AOI;
   // 19 = Uncertain, using last known good;    20 = Uncertain, using replacement value;
   // 32 = Bad, Signal Failure;   33 = Bad, Channel Fault;
   // 34 = Bad, Module / Comms Fault;   35 = Bad, Invalid Configuration
   // #####  V4.00.00  2018-06-25:  Modified to correct precedence and value of Simulated PV.  #####
   // #####  V4.00.01  2018-08-29:  Modified handling of Simulated PV and scaling config errors.  #####
   8: LBL(DoSrcQ)[XIO(Cfg_UseChanSrcQ) MOV(1,Wrk_SrcQ) ,XIC(Cfg_UseChanSrcQ) MOV(Inp_PVSrcQ,Wrk_SrcQ) ,XIC(Inp_PVUncertain) MOV(16,Wrk_SrcQ) ,XIC(Inp_PVBad) MOV(34,Wrk_SrcQ) ,XIC(Inp_Sim) MOV(10,Wrk_SrcQ) ,[XIC(Wrk_InpInfNaN) ,XIC(Sts_FailCmp) ] [XIO(Cfg_UseChanSrcQ) ,XIC(Inp_Sim) ] MOV(32,Wrk_SrcQ) ,[XIC(Err_Raw) ,XIC(Err_EU) ] MOV(35,Wrk_SrcQ) ,MOV(Wrk_SrcQ,SrcQ_IO) ];
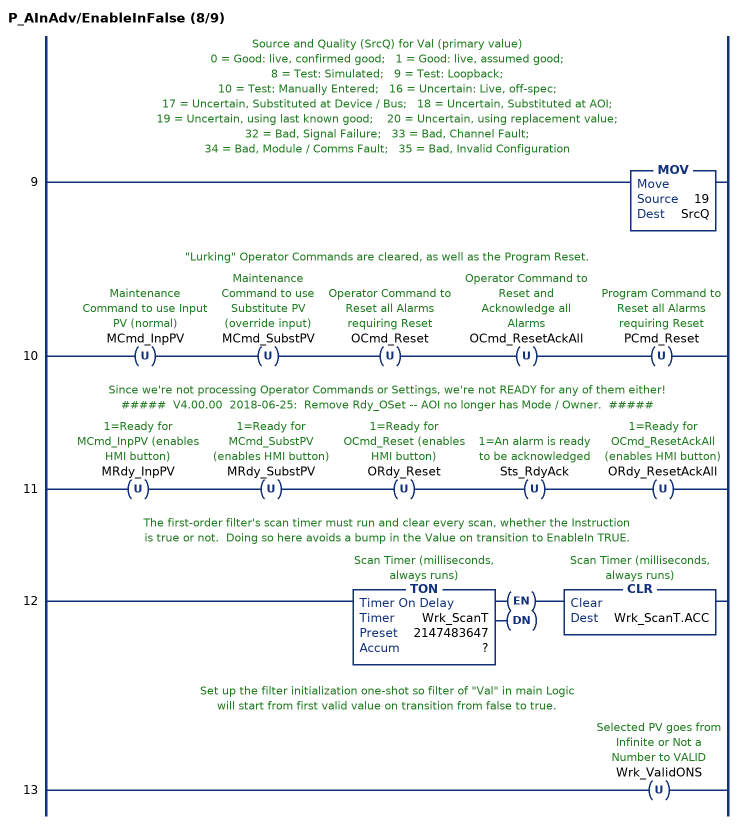
   // Source and Quality (SrcQ) for Val (primary value)
   // 0 = Good: live, confirmed good;   1 = Good: live, assumed good;
   // 8 = Test: Simulated;   9 = Test: Loopback;
   // 10 = Test: Manually Entered;   16 = Uncertain: Live, off-spec;
   // 17 = Uncertain, Substituted at Device / Bus;   18 = Uncertain, Substituted at AOI;
   // 19 = Uncertain, using last known good;    20 = Uncertain, using replacement value;
   // 32 = Bad, Signal Failure;   33 = Bad, Channel Fault;
   // 34 = Bad, Module / Comms Fault;   35 = Bad, Invalid Configuration
   9: MOV(19,SrcQ);
   // "Lurking" Operator Commands are cleared, as well as the Program Reset.
   10: OTU(MCmd_InpPV)OTU(MCmd_SubstPV)OTU(OCmd_Reset)OTU(OCmd_ResetAckAll)OTU(PCmd_Reset);
   // Since we're not processing Operator Commands or Settings, we're not READY for any of them either!
   // #####  V4.00.00  2018-06-25:  Remove Rdy_OSet -- AOI no longer has Mode / Owner.  #####
   11: OTU(MRdy_InpPV)OTU(MRdy_SubstPV)OTU(ORdy_Reset)OTU(Sts_RdyAck)OTU(ORdy_ResetAckAll);
   // The first-order filter's scan timer must run and clear every scan, whether the Instruction
   // is true or not.  Doing so here avoids a bump in the Value on transition to EnableIn TRUE.
   12: TON(Wrk_ScanT,?,?)CLR(Wrk_ScanT.ACC);
   // Set up the filter initialization one-shot so filter of "Val" in main Logic
   // will start from first valid value on transition from false to true.
   13: OTU(Wrk_ValidONS);
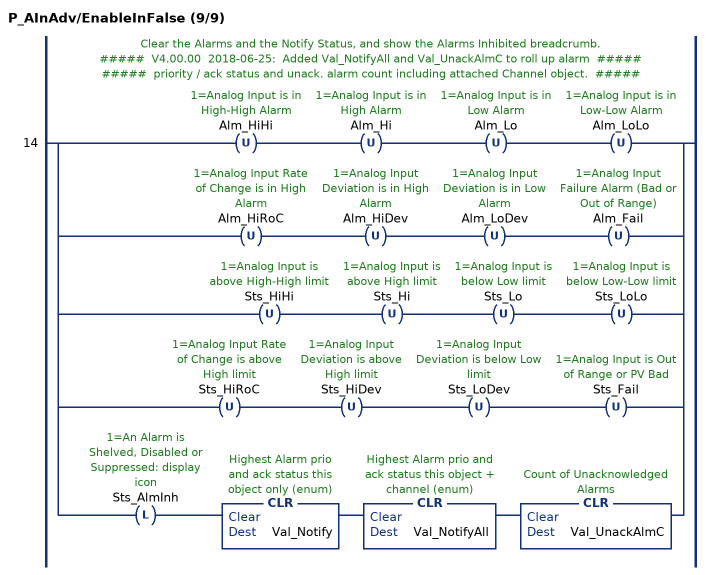
   // Clear the Alarms and the Notify Status, and show the Alarms Inhibited breadcrumb.
   // #####  V4.00.00  2018-06-25:  Added Val_NotifyAll and Val_UnackAlmC to roll up alarm  #####
   // #####  priority / ack status and unack. alarm count including attached Channel object.  #####
   14: [OTU(Alm_HiHi) OTU(Alm_Hi) OTU(Alm_Lo) OTU(Alm_LoLo) ,OTU(Alm_HiRoC) OTU(Alm_HiDev) OTU(Alm_LoDev) OTU(Alm_Fail) ,OTU(Sts_HiHi) OTU(Sts_Hi) OTU(Sts_Lo) OTU(Sts_LoLo) ,OTU(Sts_HiRoC) OTU(Sts_HiDev) OTU(Sts_LoDev) OTU(Sts_Fail) ,OTL(Sts_AlmInh) CLR(Val_Notify) CLR(Val_NotifyAll) CLR(Val_UnackAlmC) ];
END_ROUTINE

ROUTINE Logic   (* ladder *)
// Normal Scan - PV is scaled and alarms are generated
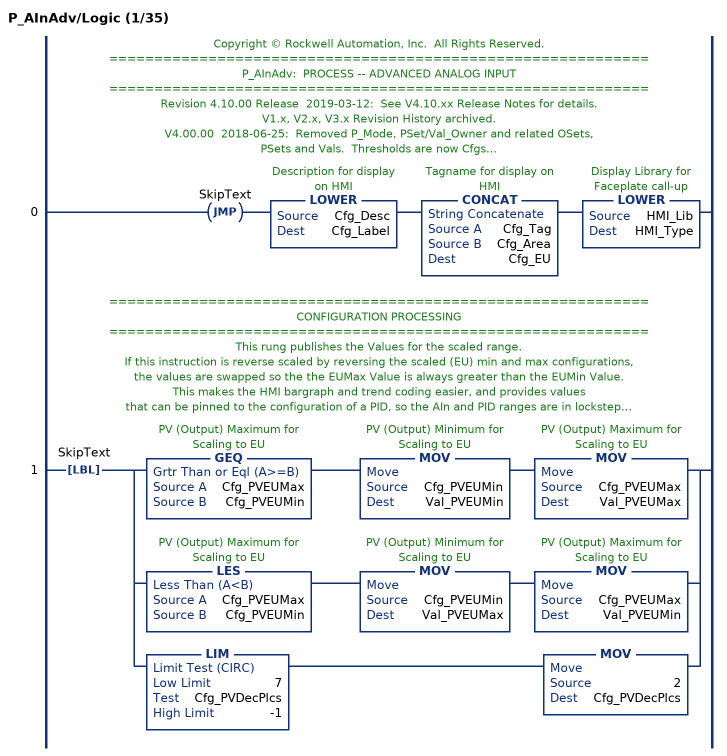
   // Copyright © Rockwell Automation, Inc.  All Rights Reserved.
   // ============================================================
   // P_AInAdv:  PROCESS -- ADVANCED ANALOG INPUT
   // ============================================================
   // Revision 4.10.00 Release  2019-03-12:  See V4.10.xx Release Notes for details.
   // V1.x, V2.x, V3.x Revision History archived.
   // V4.00.00  2018-06-25:  Removed P_Mode, PSet/Val_Owner and related OSets,
   //    PSets and Vals.  Thresholds are now Cfgs.
   // Changed Inf_ items to HMI_, and added Cfg_Area for security.
   // Added notify and unack count rollup for Channel object. Added Err_Rate.
   // Changed Out-of-Range limit checks to use raw Input (Inp_PV)
   //    instead of scaled PV (Val).  Changing EU scaling will not
   //    necessitate changing fail thresholds and deadband.
   // Deleted Cfg_PCmdClear.  All Program Commands are now self-clearing.
   // Aligned ready bit naming with command bit names.
   // All OCmds/MCmds and ORdys/MRdys are now Local Tags.
   // Added Sts_RdyAck and Sts_RdyReset for use by external objects.
   // Removed Err_DB, code ensures Status Deadband configs are always valid.
   // Added configurable decimal places for display on HMI.
   // V4.00.01  2018-08-29:  Modified handling of SrcQ_IO and SrcQ.
   // V4.10.00  2019-03-12: Added Control Limits. Added Cfg_HasMoreObj.
   // ============================================================
   // This Instruction monitors an Analog Input from a flow, level, pressure,
   // temperature, or any other analog sensor, and provides:
   // *  Scaling, from Input (Raw) to PV (Engineering) Units
   // *  High-High, High, Low and Low-Low Status and Alarms, with Gate
   // inputs and configurable on-delay, off-delay and gate delay times
   // *  Monitoring of bad/uncertain PV status, floating point exceptions
   // and out-of-range conditions, with PV Fail alarm
   // *  Setting of a simulated input signal for process simulation
   // *  Capturing of the lowest and highest PV excursion values
   // *  Configurable status thresholds, deadbands and range limits
   // *  Maintenance Commands to allow manual override of the input signal (Substitute PV)
   // **  Calculation of (filtered) signal rate of change with High Rate of Change alarm
   // **  Square Root characterization for flow scaling based on differential-pressure input
   // **  Reference (setpoint) value entry and alarms for deviation from reference (high, low)
   // ** = advanced capabilities in this instruction
   // *  = basic capabilities included in P_AIn (analog input basic) instruction
   // ============================================================
   // SHOW LOCAL STRINGS
   // ============================================================
   // The STRINGs containing the text associated with each instance of this
   // instruction cannot be Input or Output Parameters, because STRINGs are not
   //  'atomic' types. (Inputs and Outputs must be SINT, INT, DINT, REAL, or BOOL.)
   // In order to make it easier to find and configure these STRINGs, this rung
   // was added.  THE JMP (and the LBL on the following rung)
   // MUST NOT BE REMOVED!!!
   // To view the STRINGs, go to the instruction instance (in LD or FBD), RIGHT-click
   // to bring up the context menu and select "Open Instruction Logic".
   // This rung will appear with the STRING values for the selected instance.
   // You may double-click the STRING values here to modify them as well.
   // #####  V4.00-00  2018-06-25:  Added string for Cfg_Area, renamed Inf_* to HMI_*.  #####
   // #####  Removed two rungs with Mode, Owner functions.  #####
   0: JMP(SkipText)LOWER(Cfg_Desc,Cfg_Label)CONCAT(Cfg_Tag,Cfg_Area,Cfg_EU)LOWER(HMI_Lib,HMI_Type);
   // ============================================================
   // CONFIGURATION PROCESSING
   // ============================================================
   // This rung publishes the Values for the scaled range.
   // If this instruction is reverse scaled by reversing the scaled (EU) min and max configurations,
   // the values are swapped so the the EUMax Value is always greater than the EUMin Value.
   // This makes the HMI bargraph and trend coding easier, and provides values
   // that can be pinned to the configuration of a PID, so the AIn and PID ranges are in lockstep.
   // #####  V4.00.00  2018-06-25:  Added configurable decimal places for display on HMI.  #####
   1: LBL(SkipText)[GEQ(Cfg_PVEUMax,Cfg_PVEUMin) MOV(Cfg_PVEUMin,Val_PVEUMin) MOV(Cfg_PVEUMax,Val_PVEUMax) ,LES(Cfg_PVEUMax,Cfg_PVEUMin) MOV(Cfg_PVEUMin,Val_PVEUMax) MOV(Cfg_PVEUMax,Val_PVEUMin) ,LIM(7,Cfg_PVDecPlcs,-1) MOV(2,Cfg_PVDecPlcs) ];
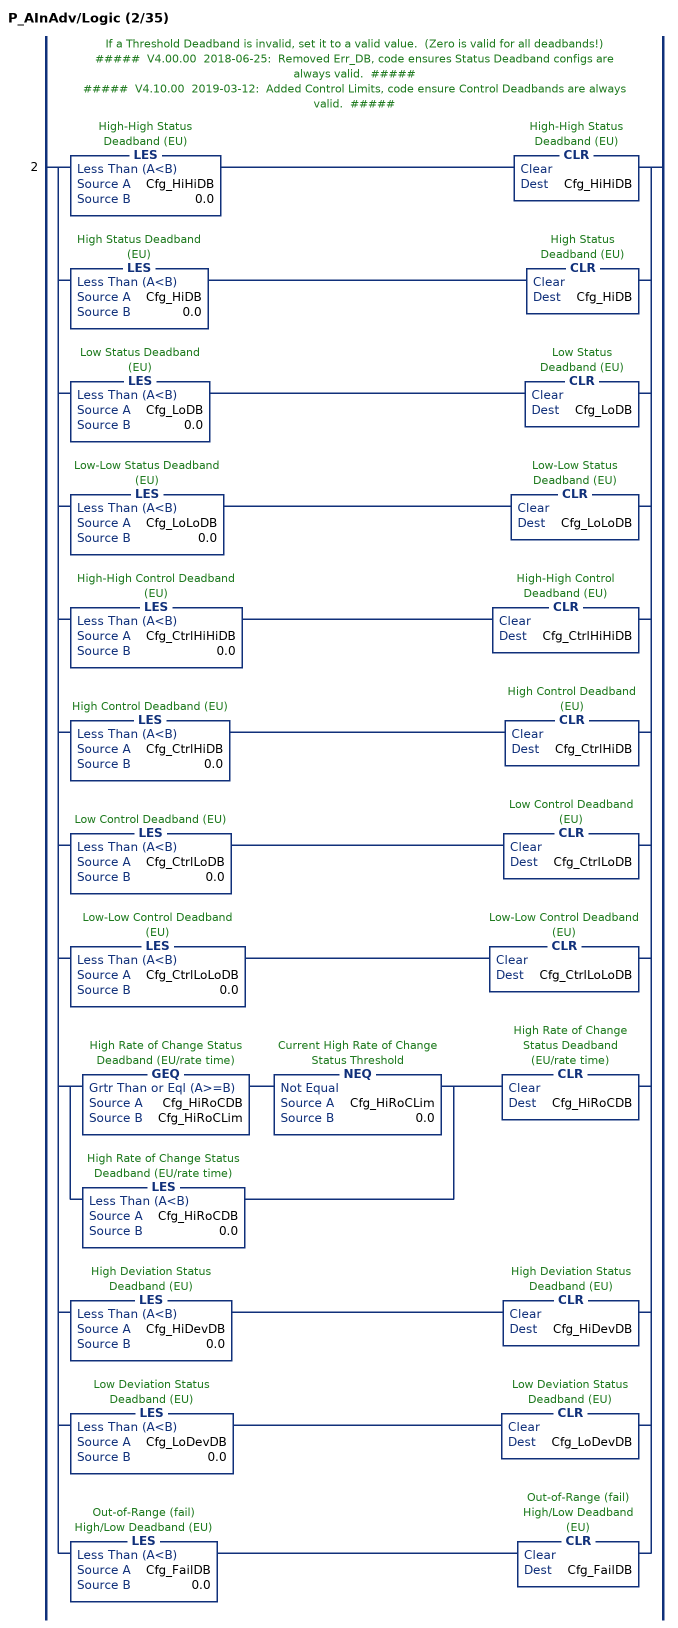
   // If a Threshold Deadband is invalid, set it to a valid value.  (Zero is valid for all deadbands!)
   // #####  V4.00.00  2018-06-25:  Removed Err_DB, code ensures Status Deadband configs are always valid.  #####
   // #####  V4.10.00  2019-03-12:  Added Control Limits, code ensure Control Deadbands are always valid.  #####
   2: [LES(Cfg_HiHiDB,0.0) CLR(Cfg_HiHiDB) ,LES(Cfg_HiDB,0.0) CLR(Cfg_HiDB) ,LES(Cfg_LoDB,0.0) CLR(Cfg_LoDB) ,LES(Cfg_LoLoDB,0.0) CLR(Cfg_LoLoDB) ,LES(Cfg_CtrlHiHiDB,0.0) CLR(Cfg_CtrlHiHiDB) ,LES(Cfg_CtrlHiDB,0.0) CLR(Cfg_CtrlHiDB) ,LES(Cfg_CtrlLoDB,0.0) CLR(Cfg_CtrlLoDB) ,LES(Cfg_CtrlLoLoDB,0.0) CLR(Cfg_CtrlLoLoDB) ,[GEQ(Cfg_HiRoCDB,Cfg_HiRoCLim) NEQ(Cfg_HiRoCLim,0.0) ,LES(Cfg_HiRoCDB,0.0) ] CLR(Cfg_HiRoCDB) ,LES(Cfg_HiDevDB,0.0) CLR(Cfg_HiDevDB) ,LES(Cfg_LoDevDB,0.0) CLR(Cfg_LoDevDB) ,LES(Cfg_FailDB,0.0) CLR(Cfg_FailDB) ];
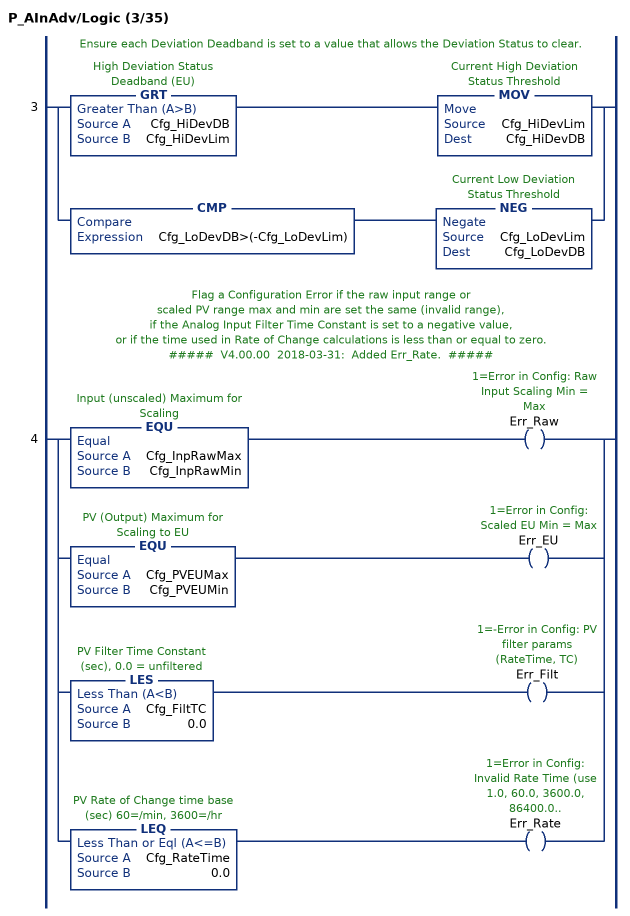
   // Ensure each Deviation Deadband is set to a value that allows the Deviation Status to clear.
   3: [GRT(Cfg_HiDevDB,Cfg_HiDevLim) MOV(Cfg_HiDevLim,Cfg_HiDevDB) ,CMP(Cfg_LoDevDB>(-Cfg_LoDevLim)) NEG(Cfg_LoDevLim,Cfg_LoDevDB) ];
   // Flag a Configuration Error if the raw input range or
   // scaled PV range max and min are set the same (invalid range),
   // if the Analog Input Filter Time Constant is set to a negative value,
   // or if the time used in Rate of Change calculations is less than or equal to zero.
   // #####  V4.00.00  2018-03-31:  Added Err_Rate.  #####
   4: [EQU(Cfg_InpRawMax,Cfg_InpRawMin) OTE(Err_Raw) ,EQU(Cfg_PVEUMax,Cfg_PVEUMin) OTE(Err_EU) ,LES(Cfg_FiltTC,0.0) OTE(Err_Filt) ,LEQ(Cfg_RateTime,0.0) OTE(Err_Rate) ];
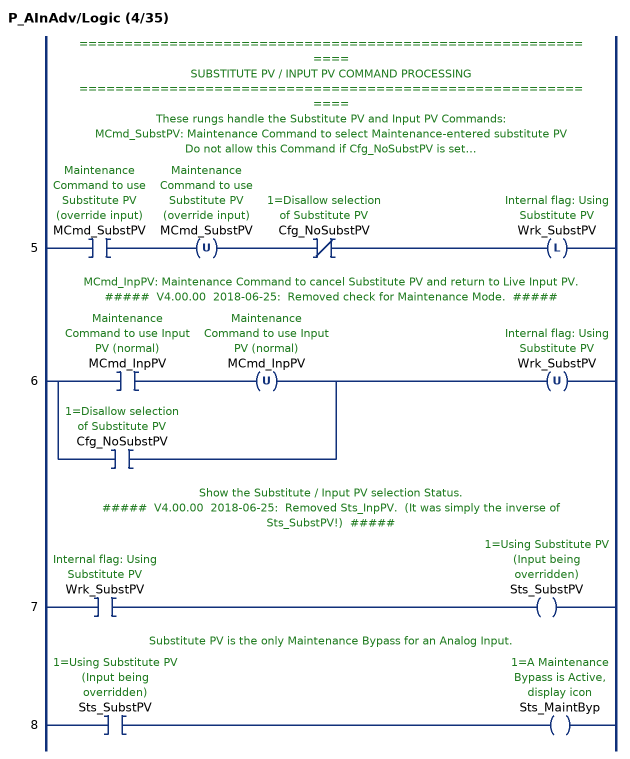
   // ============================================================
   // SUBSTITUTE PV / INPUT PV COMMAND PROCESSING
   // ============================================================
   // These rungs handle the Substitute PV and Input PV Commands:
   // MCmd_SubstPV: Maintenance Command to select Maintenance-entered substitute PV
   // Do not allow this Command if Cfg_NoSubstPV is set.
   // #####  V4.00.00  2018-06-25:  Removed check for Maintenance Mode.  #####
   5: XIC(MCmd_SubstPV)OTU(MCmd_SubstPV)XIO(Cfg_NoSubstPV)OTL(Wrk_SubstPV);
   // MCmd_InpPV: Maintenance Command to cancel Substitute PV and return to Live Input PV.
   // #####  V4.00.00  2018-06-25:  Removed check for Maintenance Mode.  #####
   6: [XIC(MCmd_InpPV) OTU(MCmd_InpPV) ,XIC(Cfg_NoSubstPV) ]OTU(Wrk_SubstPV);
   // Show the Substitute / Input PV selection Status.
   // #####  V4.00.00  2018-06-25:  Removed Sts_InpPV.  (It was simply the inverse of Sts_SubstPV!)  #####
   7: XIC(Wrk_SubstPV)OTE(Sts_SubstPV);
   // Substitute PV is the only Maintenance Bypass for an Analog Input.
   8: XIC(Sts_SubstPV)OTE(Sts_MaintByp);
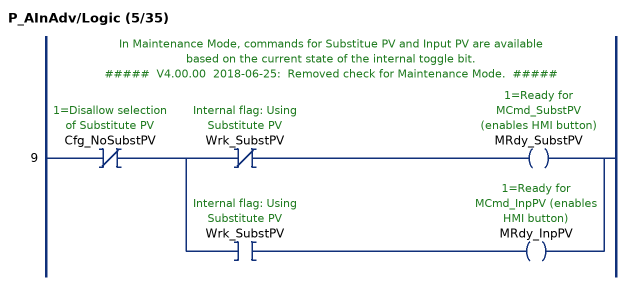
   // In Maintenance Mode, commands for Substitue PV and Input PV are available
   // based on the current state of the internal toggle bit.
   // #####  V4.00.00  2018-06-25:  Removed check for Maintenance Mode.  #####
   9: XIO(Cfg_NoSubstPV)[XIO(Wrk_SubstPV) OTE(MRdy_SubstPV) ,XIC(Wrk_SubstPV) OTE(MRdy_InpPV) ];
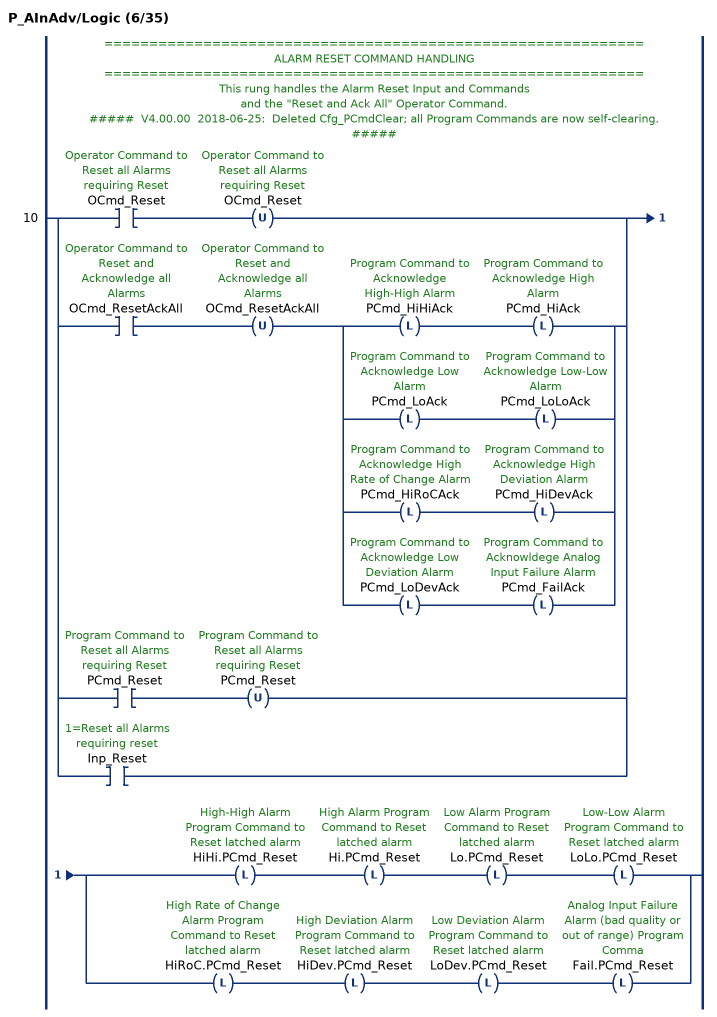
   // ============================================================
   // ALARM RESET COMMAND HANDLING
   // ============================================================
   // This rung handles the Alarm Reset Input and Commands
   // and the "Reset and Ack All" Operator Command.
   // #####  V4.00.00  2018-06-25:  Deleted Cfg_PCmdClear; all Program Commands are now self-clearing.  #####
   10: [XIC(OCmd_Reset) OTU(OCmd_Reset) ,XIC(OCmd_ResetAckAll) OTU(OCmd_ResetAckAll) [OTL(PCmd_HiHiAck) OTL(PCmd_HiAck) ,OTL(PCmd_LoAck) OTL(PCmd_LoLoAck) ,OTL(PCmd_HiRoCAck) OTL(PCmd_HiDevAck) ,OTL(PCmd_LoDevAck) OTL(PCmd_FailAck) ] ,XIC(PCmd_Reset) OTU(PCmd_Reset) ,XIC(Inp_Reset) ][OTL(HiHi.PCmd_Reset) OTL(Hi.PCmd_Reset) OTL(Lo.PCmd_Reset) OTL(LoLo.PCmd_Reset) ,OTL(HiRoC.PCmd_Reset) OTL(HiDev.PCmd_Reset) OTL(LoDev.PCmd_Reset) OTL(Fail.PCmd_Reset) ];
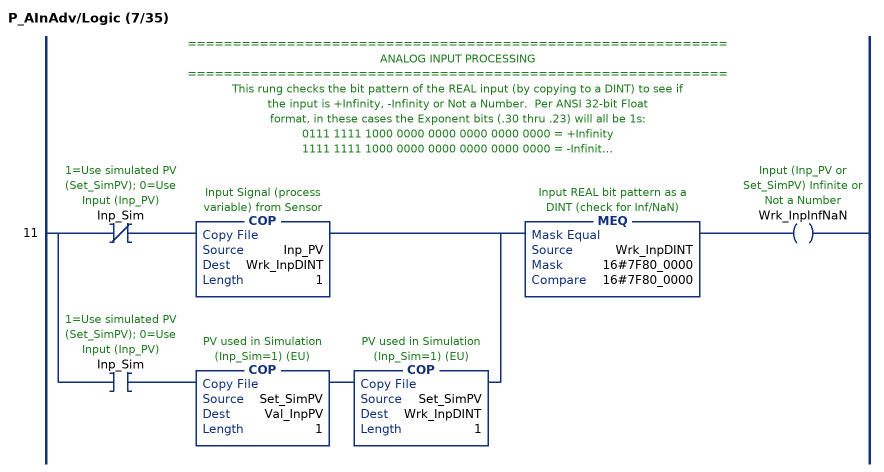
   // ============================================================
   // ANALOG INPUT PROCESSING
   // ============================================================
   // This rung checks the bit pattern of the REAL input (by copying to a DINT) to see if
   // the input is +Infinity, -Infinity or Not a Number.  Per ANSI 32-bit Float
   // format, in these cases the Exponent bits (.30 thru .23) will all be 1s:
   // 0111 1111 1000 0000 0000 0000 0000 0000 = +Infinity
   // 1111 1111 1000 0000 0000 0000 0000 0000 = -Infinity
   // x111 1111 1xxx xxxx xxxx xxxx xxxx xxxx = Not a Number
   11: [XIO(Inp_Sim) COP(Inp_PV,Wrk_InpDINT,1) ,XIC(Inp_Sim) COP(Set_SimPV,Val_InpPV,1) COP(Set_SimPV,Wrk_InpDINT,1) ]MEQ(Wrk_InpDINT,16#7F80_0000,16#7F80_0000)OTE(Wrk_InpInfNaN);
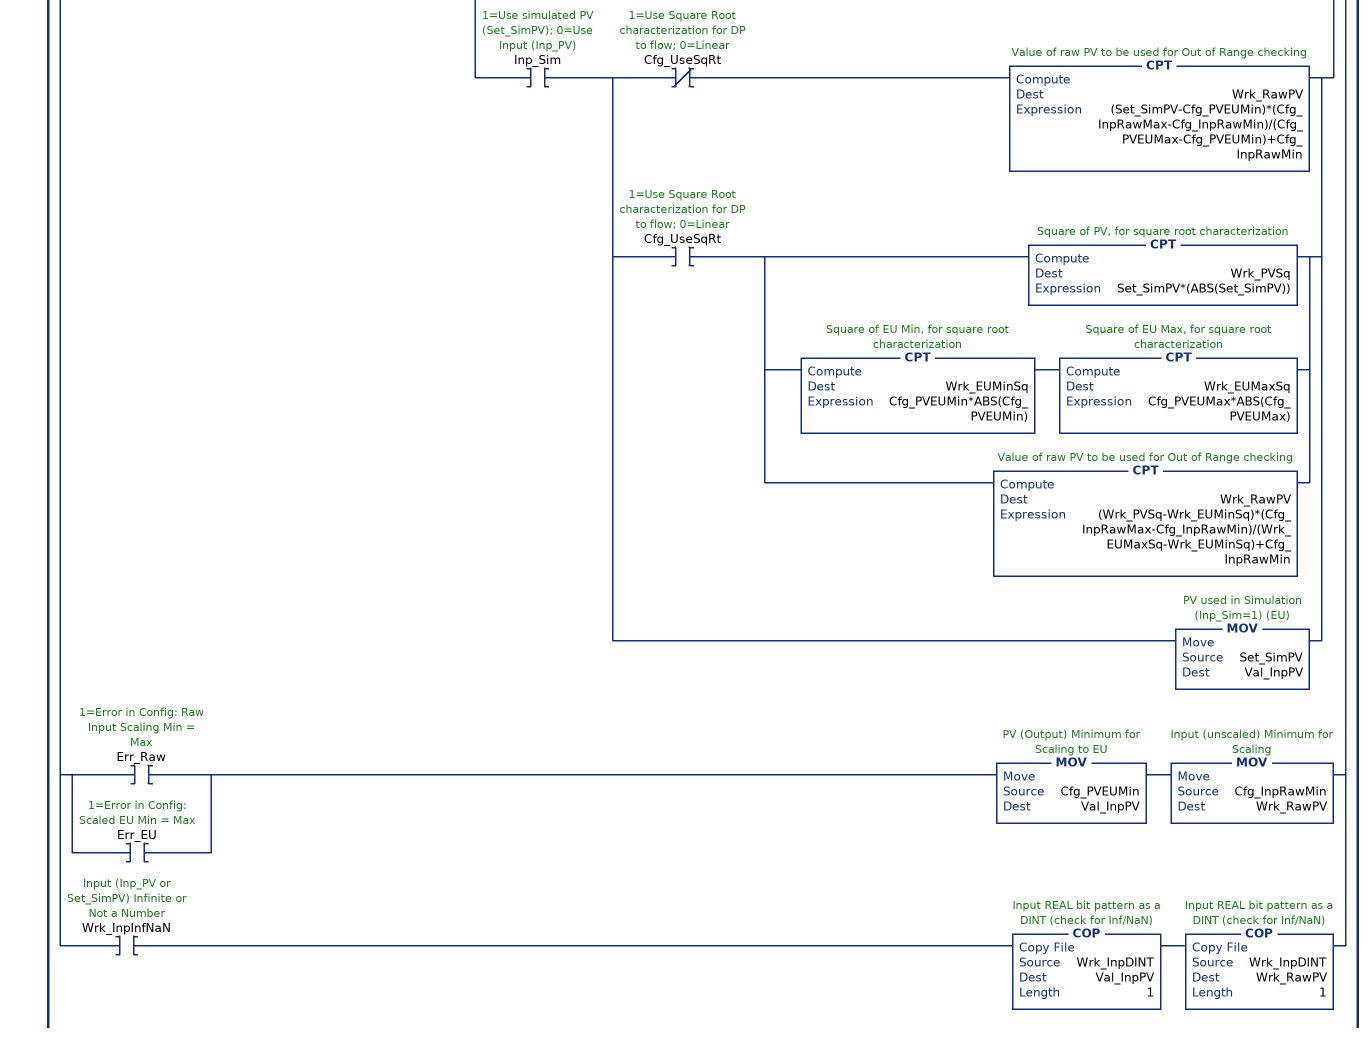
   // The Process Variable Value (Val_PV) shows the selected input,
   // regardless of Mode, EVEN WHEN EnableIn IS FALSE!
   // Here's where we select the input or the substitue PV,
   // and for the input PV, do the scaling to Engineering Units.
   // Scale to the squares of the EUMax and EUMin, then take the Square Root,
   // if the Square Root characterization is selected.  (This must work even for non-zero-based
   // inputs, say, +/- 20" WC, and show +/- flow, scaled on a square root curve each side of zero!)
   // If Square Root characterization is not selected, just do linear scaling.
   12: [XIO(Err_Raw) XIO(Err_EU) XIO(Wrk_InpInfNaN) [XIO(Inp_Sim) [XIO(Cfg_UseSqRt) CPT(Val_InpPV,(Inp_PV-Cfg_InpRawMin)*(Cfg_PVEUMax-Cfg_PVEUMin)/(Cfg_InpRawMax-Cfg_InpRawMin)+Cfg_PVEUMin) ,XIC(Cfg_UseSqRt) [CPT(Wrk_EUMinSq,Cfg_PVEUMin*ABS(Cfg_PVEUMin)) CPT(Wrk_EUMaxSq,Cfg_PVEUMax*ABS(Cfg_PVEUMax)) ,CPT(Wrk_PVSq,(Inp_PV-Cfg_InpRawMin)*(Wrk_EUMaxSq-Wrk_EUMinSq)/(Cfg_InpRawMax-Cfg_InpRawMin)+Wrk_EUMinSq) ,LES(Wrk_PVSq,0.0) CPT(Val_InpPV,-SQR(-Wrk_PVSq)) ,GEQ(Wrk_PVSq,0.0) SQR(Wrk_PVSq,Val_InpPV) ] ,MOV(Inp_PV,Wrk_RawPV) ] ,XIC(Inp_Sim) [XIO(Cfg_UseSqRt) CPT(Wrk_RawPV,(Set_SimPV-Cfg_PVEUMin)*(Cfg_InpRawMax-Cfg_InpRawMin)/(Cfg_PVEUMax-Cfg_PVEUMin)+Cfg_InpRawMin) ,XIC(Cfg_UseSqRt) [CPT(Wrk_PVSq,Set_SimPV*(ABS(Set_SimPV))) ,CPT(Wrk_EUMinSq,Cfg_PVEUMin*ABS(Cfg_PVEUMin)) CPT(Wrk_EUMaxSq,Cfg_PVEUMax*ABS(Cfg_PVEUMax)) ,CPT(Wrk_RawPV,(Wrk_PVSq-Wrk_EUMinSq)*(Cfg_InpRawMax-Cfg_InpRawMin)/(Wrk_EUMaxSq-Wrk_EUMinSq)+Cfg_InpRawMin) ] ,MOV(Set_SimPV,Val_InpPV) ] ] ,[XIC(Err_Raw) ,XIC(Err_EU) ] MOV(Cfg_PVEUMin,Val_InpPV) MOV(Cfg_InpRawMin,Wrk_RawPV) ,XIC(Wrk_InpInfNaN) COP(Wrk_InpDINT,Val_InpPV,1) COP(Wrk_InpDINT,Wrk_RawPV,1) ];
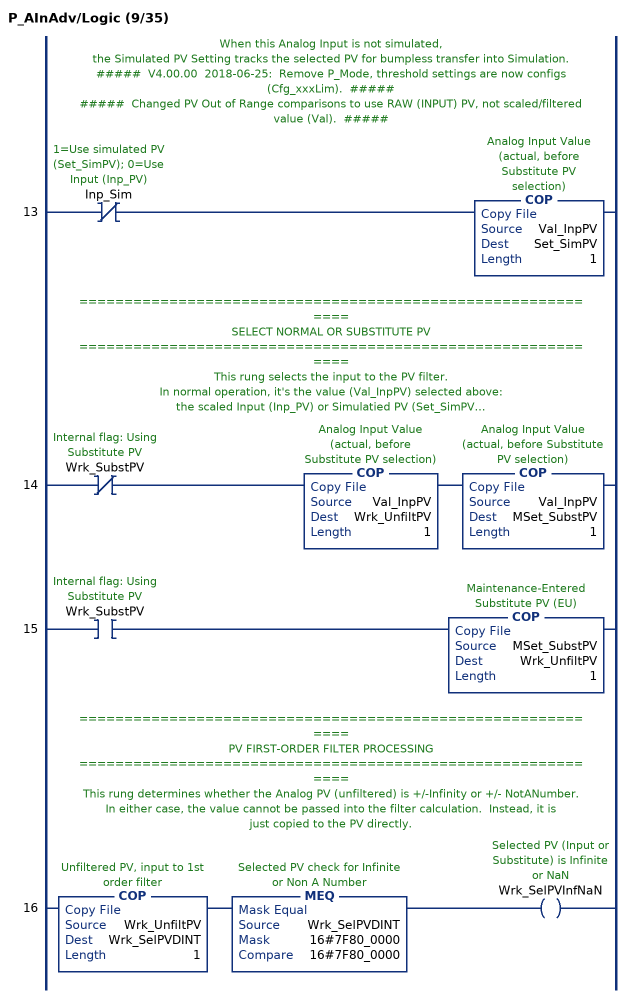
   // When this Analog Input is not simulated,
   // the Simulated PV Setting tracks the selected PV for bumpless transfer into Simulation.
   // #####  V4.00.00  2018-06-25:  Remove P_Mode, threshold settings are now configs (Cfg_xxxLim).  #####
   // #####  Changed PV Out of Range comparisons to use RAW (INPUT) PV, not scaled/filtered value (Val).  #####
   13: XIO(Inp_Sim)COP(Val_InpPV,Set_SimPV,1);
   // ============================================================
   // SELECT NORMAL OR SUBSTITUTE PV
   // ============================================================
   // This rung selects the input to the PV filter.
   // In normal operation, it's the value (Val_InpPV) selected above:
   // the scaled Input (Inp_PV) or Simulatied PV (Set_SimPV)
   // (and this value tracks back into the Substitute PV setting).
   // With Substitute PV enabled, it's the value of the entered MSet_SubstPV.
   14: XIO(Wrk_SubstPV)COP(Val_InpPV,Wrk_UnfiltPV,1)COP(Val_InpPV,MSet_SubstPV,1);
   15: XIC(Wrk_SubstPV)COP(MSet_SubstPV,Wrk_UnfiltPV,1);
   // ============================================================
   // PV FIRST-ORDER FILTER PROCESSING
   // ============================================================
   // This rung determines whether the Analog PV (unfiltered) is +/-Infinity or +/- NotANumber.
   // In either case, the value cannot be passed into the filter calculation.  Instead, it is
   // just copied to the PV directly.
   16: COP(Wrk_UnfiltPV,Wrk_SelPVDINT,1)MEQ(Wrk_SelPVDINT,16#7F80_0000,16#7F80_0000)OTE(Wrk_SelPVInfNaN);
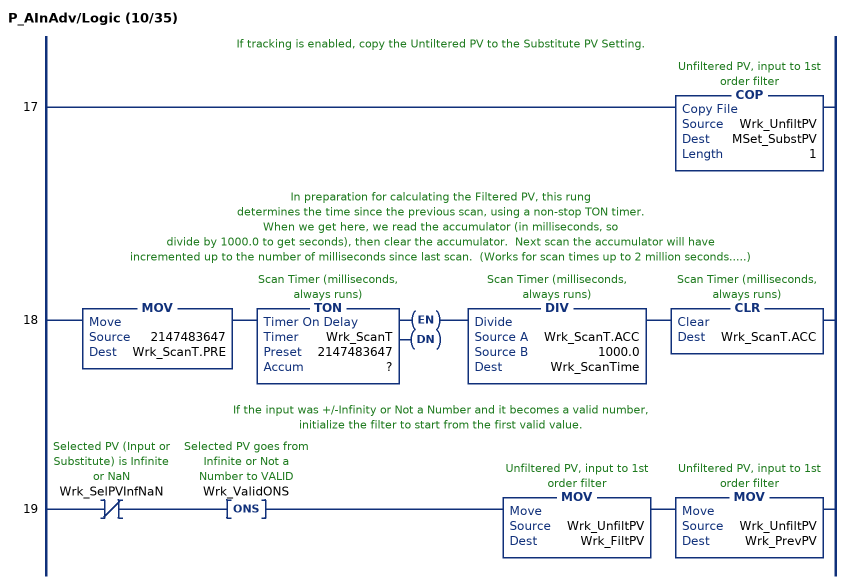
   // If tracking is enabled, copy the Untiltered PV to the Substitute PV Setting.
   17: COP(Wrk_UnfiltPV,MSet_SubstPV,1);
   // In preparation for calculating the Filtered PV, this rung
   // determines the time since the previous scan, using a non-stop TON timer.
   // When we get here, we read the accumulator (in milliseconds, so
   // divide by 1000.0 to get seconds), then clear the accumulator.  Next scan the accumulator will have
   // incremented up to the number of milliseconds since last scan.  (Works for scan times up to 2 million seconds.....)
   18: MOV(2147483647,Wrk_ScanT.PRE)TON(Wrk_ScanT,?,?)DIV(Wrk_ScanT.ACC,1000.0,Wrk_ScanTime)CLR(Wrk_ScanT.ACC);
   // If the input was +/-Infinity or Not a Number and it becomes a valid number,
   // initialize the filter to start from the first valid value.
   19: XIO(Wrk_SelPVInfNaN)ONS(Wrk_ValidONS)MOV(Wrk_UnfiltPV,Wrk_FiltPV)MOV(Wrk_UnfiltPV,Wrk_PrevPV);
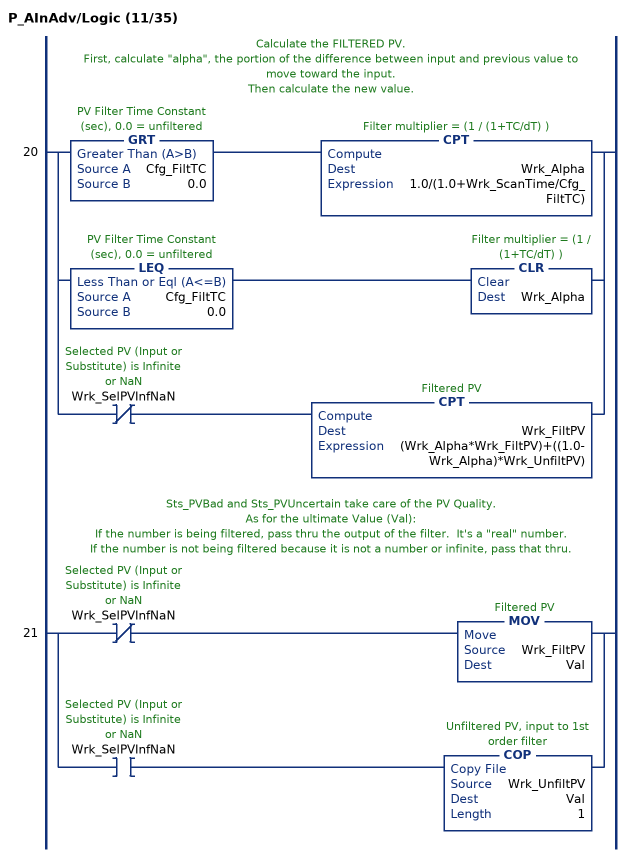
   // Calculate the FILTERED PV.
   // First, calculate "alpha", the portion of the difference between input and previous value to move toward the input.
   // Then calculate the new value.
   20: [GRT(Cfg_FiltTC,0.0) CPT(Wrk_Alpha,1.0/(1.0+Wrk_ScanTime/Cfg_FiltTC)) ,LEQ(Cfg_FiltTC,0.0) CLR(Wrk_Alpha) ,XIO(Wrk_SelPVInfNaN) CPT(Wrk_FiltPV,(Wrk_Alpha*Wrk_FiltPV)+((1.0-Wrk_Alpha)*Wrk_UnfiltPV)) ];
   // Sts_PVBad and Sts_PVUncertain take care of the PV Quality.
   // As for the ultimate Value (Val):
   // If the number is being filtered, pass thru the output of the filter.  It's a "real" number.
   // If the number is not being filtered because it is not a number or infinite, pass that thru.
   21: [XIO(Wrk_SelPVInfNaN) MOV(Wrk_FiltPV,Val) ,XIC(Wrk_SelPVInfNaN) COP(Wrk_UnfiltPV,Val,1) ];
